Yaskawa INFORM job: DEMO_NAIHAN_0625_2PAINT_1.JBI

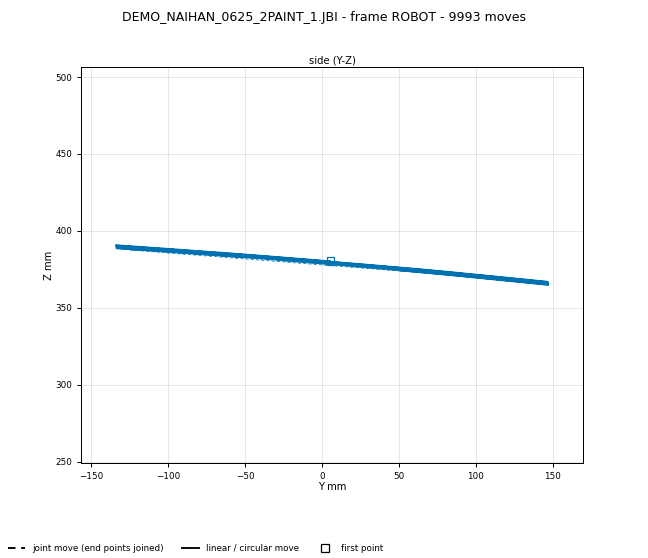
[picture p0: tool path of DEMO_NAIHAN_0625_2PAINT_1.JBI in frame ROBOT, 9993 of 9993 moves have a stored position in this frame; points joined in program order, loops and branches not executed]
/JOB
//NAME DEMO_NAIHAN_0625_2PAINT1
//POS
///NPOS 9993,0,0,0,0,0
///TOOL 1
///USER 0
///POSTYPE ROBOT
///RECTAN
///RCONF 1,0,0,0,1,0,0,0,0,0,0,0,0,0,0,0,0,0,0,0,0,0,0,0
C00000=1015.716,5.571,380.559,-24.182,21.519,-42.786
C00001=1015.718,5.240,380.586,-24.181,21.518,-42.792
C00002=1015.721,4.909,380.612,-24.181,21.519,-42.795
C00003=1015.723,4.578,380.640,-24.180,21.519,-42.799
C00004=1015.725,4.247,380.667,-24.180,21.521,-42.803
C00005=1015.727,3.917,380.694,-24.179,21.520,-42.807
C00006=1015.730,3.604,380.720,-24.179,21.521,-42.810
C00007=1015.732,3.315,380.744,-24.179,21.521,-42.814
C00008=1015.733,3.046,380.766,-24.178,21.522,-42.818
C00009=1015.736,2.783,380.787,-24.177,21.522,-42.823
C00010=1015.737,2.515,380.809,-24.177,21.522,-42.827
C00011=1015.740,2.226,380.832,-24.176,21.523,-42.831
C00012=1015.741,1.915,380.858,-24.176,21.523,-42.834
C00013=1015.744,1.584,380.885,-24.175,21.523,-42.838
C00014=1015.746,1.250,380.912,-24.175,21.524,-42.842
C00015=1015.749,0.917,380.940,-24.174,21.525,-42.846
C00016=1015.750,0.582,380.967,-24.173,21.525,-42.851
C00017=1015.752,0.246,380.994,-24.173,21.525,-42.855
C00018=1015.754,-0.092,381.021,-24.172,21.526,-42.858
C00019=1015.756,-0.430,381.049,-24.172,21.526,-42.864
C00020=1015.759,-0.771,381.077,-24.171,21.526,-42.867
C00021=1015.761,-1.112,381.105,-24.170,21.527,-42.873
C00022=1015.763,-1.455,381.132,-24.170,21.527,-42.877
C00023=1015.766,-1.801,381.161,-24.169,21.528,-42.880
C00024=1015.768,-2.146,381.188,-24.169,21.528,-42.886
C00025=1015.770,-2.495,381.217,-24.168,21.529,-42.890
C00026=1015.772,-2.845,381.245,-24.167,21.529,-42.895
C00027=1015.774,-3.196,381.274,-24.167,21.529,-42.899
C00028=1015.776,-3.549,381.302,-24.166,21.529,-42.904
C00029=1015.778,-3.903,381.331,-24.166,21.531,-42.908
C00030=1015.780,-4.260,381.360,-24.165,21.530,-42.913
C00031=1015.782,-4.622,381.389,-24.164,21.531,-42.919
C00032=1015.784,-4.988,381.419,-24.164,21.532,-42.923
C00033=1015.787,-5.358,381.448,-24.163,21.532,-42.928
C00034=1015.789,-5.732,381.479,-24.163,21.533,-42.932
C00035=1015.791,-6.107,381.510,-24.162,21.533,-42.937
C00036=1015.793,-6.483,381.540,-24.161,21.533,-42.941
C00037=1015.795,-6.858,381.571,-24.160,21.534,-42.947
C00038=1015.797,-7.229,381.601,-24.160,21.534,-42.952
C00039=1015.798,-7.598,381.630,-24.159,21.535,-42.956
C00040=1015.801,-7.964,381.660,-24.158,21.535,-42.961
C00041=1015.802,-8.327,381.689,-24.158,21.536,-42.967
C00042=1015.804,-8.690,381.719,-24.157,21.536,-42.971
C00043=1015.806,-9.053,381.748,-24.156,21.536,-42.976
C00044=1015.808,-9.416,381.776,-24.156,21.537,-42.982
C00045=1015.810,-9.778,381.806,-24.155,21.538,-42.985
C00046=1015.811,-10.139,381.835,-24.154,21.538,-42.991
C00047=1015.814,-10.500,381.865,-24.154,21.539,-42.995
C00048=1015.815,-10.860,381.893,-24.153,21.539,-43.000
C00049=1015.816,-11.219,381.922,-24.152,21.539,-43.006
C00050=1015.819,-11.577,381.950,-24.152,21.540,-43.009
C00051=1015.821,-11.933,381.980,-24.151,21.540,-43.014
C00052=1015.822,-12.288,382.008,-24.151,21.541,-43.019
C00053=1015.823,-12.641,382.036,-24.150,21.541,-43.024
C00054=1015.825,-12.993,382.065,-24.149,21.542,-43.028
C00055=1015.826,-13.344,382.093,-24.149,21.542,-43.033
C00056=1015.828,-13.692,382.121,-24.148,21.543,-43.037
C00057=1015.830,-14.038,382.149,-24.147,21.543,-43.042
C00058=1015.831,-14.383,382.176,-24.147,21.544,-43.046
C00059=1015.832,-14.725,382.203,-24.146,21.544,-43.052
C00060=1015.834,-15.065,382.230,-24.146,21.544,-43.055
C00061=1015.836,-15.402,382.257,-24.145,21.545,-43.061
C00062=1015.837,-15.739,382.285,-24.145,21.546,-43.065
C00063=1015.838,-16.075,382.311,-24.144,21.546,-43.070
C00064=1015.840,-16.408,382.337,-24.143,21.546,-43.074
C00065=1015.841,-16.742,382.364,-24.142,21.547,-43.079
C00066=1015.842,-17.075,382.391,-24.142,21.547,-43.083
C00067=1015.843,-17.409,382.417,-24.141,21.547,-43.088
C00068=1015.845,-17.742,382.444,-24.141,21.548,-43.092
C00069=1015.846,-18.107,382.474,-24.140,21.549,-43.100
C00070=1015.847,-18.329,382.491,-24.139,21.548,-43.103
C00071=1015.848,-18.576,382.510,-24.139,21.549,-43.105
C00072=1015.849,-18.837,382.531,-24.139,21.550,-43.107
C00073=1015.850,-19.099,382.552,-24.139,21.550,-43.109
C00074=1015.851,-19.347,382.573,-24.138,21.550,-43.112
C00075=1015.852,-19.764,382.605,-24.137,21.550,-43.118
C00076=1015.853,-19.936,382.619,-24.137,21.551,-43.122
C00077=1015.854,-20.269,382.646,-24.136,21.551,-43.127
C00078=1015.855,-20.602,382.672,-24.136,21.552,-43.131
C00079=1015.856,-20.934,382.698,-24.135,21.553,-43.135
C00080=1015.857,-21.267,382.725,-24.134,21.552,-43.140
C00081=1015.859,-21.599,382.751,-24.134,21.553,-43.144
C00082=1015.860,-21.933,382.777,-24.133,21.554,-43.149
C00083=1015.861,-22.265,382.804,-24.133,21.554,-43.153
C00084=1015.862,-22.598,382.831,-24.132,21.554,-43.158
C00085=1015.862,-22.930,382.857,-24.131,21.556,-43.162
C00086=1015.864,-23.264,382.883,-24.131,21.555,-43.168
C00087=1015.864,-23.596,382.909,-24.130,21.556,-43.171
C00088=1015.866,-23.929,382.936,-24.129,21.556,-43.177
C00089=1015.866,-24.262,382.962,-24.129,21.557,-43.181
C00090=1015.868,-24.595,382.989,-24.128,21.557,-43.186
C00091=1015.868,-24.928,383.015,-24.128,21.558,-43.190
C00092=1015.869,-25.260,383.041,-24.127,21.558,-43.195
C00093=1015.870,-25.594,383.067,-24.126,21.559,-43.199
C00094=1015.871,-25.926,383.094,-24.126,21.559,-43.204
C00095=1015.871,-26.259,383.120,-24.125,21.559,-43.208
C00096=1015.873,-26.592,383.147,-24.124,21.560,-43.214
C00097=1015.874,-26.924,383.172,-24.124,21.560,-43.217
C00098=1015.875,-27.256,383.198,-24.123,21.560,-43.223
C00099=1015.875,-27.589,383.225,-24.123,21.562,-43.227
C00100=1015.877,-27.922,383.251,-24.122,21.562,-43.232
C00101=1015.877,-28.255,383.277,-24.121,21.562,-43.236
C00102=1015.878,-28.587,383.303,-24.120,21.562,-43.241
C00103=1015.878,-28.920,383.330,-24.120,21.563,-43.245
C00104=1015.879,-29.253,383.355,-24.119,21.563,-43.250
C00105=1015.879,-29.586,383.381,-24.119,21.564,-43.254
C00106=1015.881,-29.918,383.408,-24.118,21.565,-43.260
C00107=1015.882,-30.252,383.434,-24.118,21.565,-43.264
C00108=1015.882,-30.584,383.460,-24.117,21.565,-43.269
C00109=1015.883,-30.917,383.486,-24.116,21.566,-43.273
C00110=1015.883,-31.250,383.512,-24.116,21.566,-43.278
C00111=1015.884,-31.582,383.538,-24.115,21.567,-43.282
C00112=1015.884,-31.915,383.565,-24.114,21.567,-43.287
C00113=1015.885,-32.248,383.590,-24.114,21.568,-43.291
C00114=1015.885,-32.581,383.617,-24.113,21.568,-43.296
C00115=1015.886,-32.914,383.643,-24.113,21.569,-43.301
C00116=1015.886,-33.247,383.668,-24.112,21.569,-43.306
C00117=1015.886,-33.579,383.694,-24.111,21.570,-43.310
C00118=1015.887,-33.912,383.721,-24.111,21.570,-43.315
C00119=1015.888,-34.245,383.746,-24.110,21.571,-43.319
C00120=1015.888,-34.577,383.772,-24.109,21.571,-43.324
C00121=1015.889,-34.910,383.799,-24.109,21.572,-43.328
C00122=1015.889,-35.243,383.824,-24.108,21.572,-43.334
C00123=1015.889,-35.575,383.850,-24.108,21.573,-43.337
C00124=1015.890,-35.908,383.876,-24.107,21.573,-43.343
C00125=1015.890,-36.241,383.902,-24.107,21.574,-43.347
C00126=1015.890,-36.573,383.928,-24.106,21.574,-43.352
C00127=1015.891,-36.905,383.954,-24.105,21.574,-43.357
C00128=1015.892,-37.239,383.979,-24.105,21.575,-43.361
C00129=1015.891,-37.571,384.005,-24.104,21.575,-43.366
C00130=1015.892,-37.903,384.031,-24.103,21.576,-43.371
C00131=1015.893,-38.236,384.057,-24.102,21.576,-43.376
C00132=1015.892,-38.569,384.083,-24.102,21.577,-43.380
C00133=1015.892,-38.902,384.109,-24.101,21.577,-43.385
C00134=1015.892,-39.235,384.134,-24.101,21.578,-43.389
C00135=1015.893,-39.567,384.161,-24.100,21.578,-43.394
C00136=1015.893,-39.899,384.186,-24.100,21.579,-43.398
C00137=1015.894,-40.233,384.212,-24.099,21.579,-43.404
C00138=1015.893,-40.565,384.237,-24.098,21.580,-43.409
C00139=1015.894,-40.897,384.264,-24.098,21.580,-43.413
C00140=1015.894,-41.230,384.289,-24.097,21.580,-43.418
C00141=1015.894,-41.562,384.314,-24.096,21.582,-43.422
C00142=1015.894,-41.895,384.341,-24.096,21.582,-43.427
C00143=1015.894,-42.228,384.366,-24.095,21.582,-43.431
C00144=1015.893,-42.561,384.392,-24.094,21.583,-43.437
C00145=1015.894,-42.893,384.418,-24.094,21.583,-43.442
C00146=1015.894,-43.226,384.443,-24.093,21.583,-43.446
C00147=1015.894,-43.558,384.469,-24.092,21.584,-43.451
C00148=1015.894,-43.890,384.494,-24.092,21.585,-43.455
C00149=1015.894,-44.223,384.520,-24.091,21.585,-43.461
C00150=1015.894,-44.556,384.546,-24.091,21.586,-43.465
C00151=1015.894,-44.888,384.571,-24.090,21.586,-43.470
C00152=1015.894,-45.221,384.596,-24.089,21.586,-43.475
C00153=1015.893,-45.554,384.622,-24.089,21.587,-43.479
C00154=1015.893,-45.886,384.647,-24.088,21.588,-43.485
C00155=1015.893,-46.219,384.673,-24.088,21.588,-43.488
C00156=1015.893,-46.551,384.699,-24.087,21.588,-43.494
C00157=1015.894,-46.884,384.724,-24.086,21.590,-43.498
C00158=1015.893,-47.216,384.750,-24.086,21.589,-43.503
C00159=1015.893,-47.548,384.776,-24.085,21.589,-43.508
C00160=1015.892,-47.881,384.800,-24.084,21.591,-43.512
C00161=1015.892,-48.213,384.826,-24.083,21.591,-43.518
C00162=1015.891,-48.546,384.852,-24.083,21.592,-43.522
C00163=1015.892,-48.879,384.877,-24.082,21.592,-43.527
C00164=1015.891,-49.211,384.902,-24.081,21.592,-43.532
C00165=1015.891,-49.543,384.928,-24.081,21.593,-43.536
C00166=1015.891,-49.876,384.953,-24.080,21.593,-43.542
C00167=1015.891,-50.208,384.979,-24.080,21.595,-43.546
C00168=1015.890,-50.540,385.004,-24.079,21.594,-43.551
C00169=1015.890,-50.873,385.029,-24.079,21.595,-43.555
C00170=1015.890,-51.205,385.055,-24.078,21.596,-43.560
C00171=1015.890,-51.537,385.080,-24.077,21.596,-43.566
C00172=1015.889,-51.870,385.105,-24.077,21.597,-43.570
C00173=1015.888,-52.203,385.131,-24.076,21.597,-43.575
C00174=1015.888,-52.535,385.156,-24.075,21.597,-43.579
C00175=1015.887,-52.867,385.181,-24.075,21.598,-43.584
C00176=1015.887,-53.200,385.206,-24.074,21.598,-43.589
C00177=1015.886,-53.532,385.231,-24.074,21.600,-43.594
C00178=1015.886,-53.864,385.257,-24.073,21.599,-43.599
C00179=1015.885,-54.196,385.282,-24.072,21.600,-43.603
C00180=1015.885,-54.528,385.307,-24.072,21.601,-43.608
C00181=1015.884,-54.860,385.332,-24.071,21.601,-43.613
C00182=1015.884,-55.193,385.357,-24.070,21.602,-43.618
C00183=1015.882,-55.526,385.383,-24.070,21.602,-43.623
C00184=1015.882,-55.859,385.408,-24.069,21.603,-43.627
C00185=1015.882,-56.191,385.434,-24.068,21.603,-43.632
C00186=1015.881,-56.524,385.458,-24.068,21.603,-43.637
C00187=1015.880,-56.858,385.484,-24.067,21.605,-43.642
C00188=1015.880,-57.191,385.509,-24.066,21.604,-43.647
C00189=1015.879,-57.524,385.534,-24.066,21.605,-43.652
C00190=1015.878,-57.858,385.559,-24.065,21.606,-43.656
C00191=1015.877,-58.193,385.584,-24.064,21.606,-43.662
C00192=1015.876,-58.527,385.610,-24.064,21.607,-43.666
C00193=1015.876,-58.862,385.635,-24.063,21.607,-43.671
C00194=1015.875,-59.197,385.660,-24.062,21.608,-43.676
C00195=1015.874,-59.533,385.686,-24.062,21.608,-43.680
C00196=1015.874,-59.869,385.711,-24.061,21.609,-43.686
C00197=1015.873,-60.206,385.736,-24.060,21.609,-43.691
C00198=1015.872,-60.543,385.761,-24.060,21.610,-43.695
C00199=1015.871,-60.880,385.787,-24.059,21.610,-43.700
C00200=1015.870,-61.217,385.812,-24.059,21.611,-43.706
C00201=1015.869,-61.555,385.837,-24.058,21.611,-43.710
C00202=1015.868,-61.894,385.863,-24.057,21.612,-43.715
C00203=1015.867,-62.232,385.888,-24.057,21.612,-43.720
C00204=1015.867,-62.571,385.914,-24.056,21.614,-43.725
C00205=1015.865,-62.911,385.939,-24.055,21.613,-43.730
C00206=1015.864,-63.251,385.965,-24.055,21.614,-43.735
C00207=1015.863,-63.592,385.990,-24.054,21.615,-43.739
C00208=1015.862,-63.933,386.016,-24.053,21.616,-43.745
C00209=1015.861,-64.273,386.041,-24.053,21.615,-43.750
C00210=1015.860,-64.614,386.067,-24.052,21.617,-43.754
C00211=1015.859,-64.956,386.092,-24.051,21.617,-43.759
C00212=1015.857,-65.298,386.118,-24.051,21.618,-43.765
C00213=1015.857,-65.640,386.144,-24.050,21.617,-43.770
C00214=1015.855,-65.983,386.169,-24.050,21.619,-43.774
C00215=1015.854,-66.325,386.195,-24.049,21.619,-43.780
C00216=1015.853,-66.667,386.220,-24.048,21.620,-43.785
C00217=1015.852,-67.011,386.246,-24.048,21.620,-43.789
C00218=1015.850,-67.354,386.271,-24.047,21.621,-43.795
C00219=1015.849,-67.697,386.297,-24.046,21.621,-43.800
C00220=1015.848,-68.041,386.323,-24.045,21.622,-43.805
C00221=1015.846,-68.384,386.348,-24.045,21.622,-43.809
C00222=1015.845,-68.728,386.373,-24.044,21.623,-43.815
C00223=1015.844,-69.072,386.399,-24.043,21.623,-43.820
C00224=1015.843,-69.416,386.425,-24.043,21.624,-43.824
C00225=1015.841,-69.759,386.450,-24.042,21.624,-43.829
C00226=1015.840,-70.104,386.475,-24.041,21.625,-43.835
C00227=1015.838,-70.448,386.501,-24.041,21.625,-43.840
C00228=1015.837,-70.792,386.527,-24.040,21.626,-43.844
C00229=1015.835,-71.136,386.552,-24.040,21.627,-43.850
C00230=1015.834,-71.481,386.577,-24.039,21.627,-43.855
C00231=1015.832,-71.825,386.603,-24.038,21.628,-43.861
C00232=1015.830,-72.168,386.628,-24.038,21.628,-43.865
C00233=1015.829,-72.512,386.654,-24.037,21.629,-43.870
C00234=1015.827,-72.856,386.679,-24.036,21.629,-43.875
C00235=1015.826,-73.200,386.705,-24.035,21.630,-43.881
C00236=1015.824,-73.544,386.729,-24.035,21.630,-43.885
C00237=1015.823,-73.888,386.755,-24.034,21.631,-43.890
C00238=1015.821,-74.232,386.780,-24.033,21.632,-43.896
C00239=1015.820,-74.575,386.806,-24.033,21.632,-43.901
C00240=1015.818,-74.919,386.831,-24.032,21.633,-43.905
C00241=1015.816,-75.262,386.857,-24.031,21.633,-43.911
C00242=1015.814,-75.605,386.882,-24.031,21.634,-43.916
C00243=1015.812,-75.949,386.907,-24.030,21.634,-43.920
C00244=1015.810,-76.291,386.932,-24.030,21.635,-43.926
C00245=1015.809,-76.634,386.957,-24.029,21.635,-43.931
C00246=1015.807,-76.976,386.983,-24.028,21.636,-43.936
C00247=1015.805,-77.318,387.008,-24.028,21.636,-43.940
C00248=1015.804,-77.661,387.032,-24.027,21.637,-43.946
C00249=1015.801,-78.002,387.058,-24.026,21.637,-43.951
C00250=1015.800,-78.344,387.083,-24.026,21.639,-43.955
C00251=1015.798,-78.685,387.108,-24.025,21.638,-43.960
C00252=1015.796,-79.026,387.133,-24.024,21.639,-43.966
C00253=1015.794,-79.366,387.157,-24.023,21.639,-43.971
C00254=1015.792,-79.707,387.183,-24.023,21.641,-43.975
C00255=1015.790,-80.046,387.208,-24.022,21.641,-43.981
C00256=1015.788,-80.386,387.233,-24.021,21.641,-43.986
C00257=1015.786,-80.724,387.257,-24.021,21.643,-43.990
C00258=1015.784,-81.064,387.281,-24.020,21.643,-43.995
C00259=1015.782,-81.402,387.306,-24.020,21.643,-44.001
C00260=1015.780,-81.739,387.331,-24.019,21.644,-44.005
C00261=1015.778,-82.077,387.356,-24.018,21.645,-44.010
C00262=1015.776,-82.414,387.380,-24.018,21.645,-44.016
C00263=1015.773,-82.750,387.405,-24.017,21.645,-44.021
C00264=1015.771,-83.086,387.429,-24.016,21.646,-44.025
C00265=1015.769,-83.422,387.453,-24.016,21.647,-44.031
C00266=1015.767,-83.758,387.477,-24.015,21.647,-44.036
C00267=1015.765,-84.093,387.502,-24.015,21.648,-44.040
C00268=1015.763,-84.426,387.527,-24.014,21.648,-44.045
C00269=1015.760,-84.777,387.552,-24.013,21.649,-44.051
C00270=1015.758,-85.174,387.581,-24.012,21.650,-44.056
C00271=1015.757,-85.386,387.597,-24.012,21.649,-44.060
C00272=1015.755,-85.600,387.612,-24.012,21.649,-44.062
C00273=1015.752,-86.008,387.642,-24.011,21.650,-44.067
C00274=1015.750,-86.367,387.668,-24.010,21.651,-44.073
C00275=1015.747,-86.697,387.692,-24.009,21.652,-44.078
C00276=1015.745,-87.019,387.715,-24.009,21.652,-44.082
C00277=1015.743,-87.336,387.738,-24.008,21.653,-44.088
C00278=1015.741,-87.648,387.760,-24.007,21.653,-44.093
C00279=1015.738,-87.959,387.783,-24.007,21.654,-44.097
C00280=1015.736,-88.271,387.806,-24.006,21.654,-44.102
C00281=1015.734,-88.590,387.828,-24.006,21.655,-44.106
C00282=1015.731,-88.961,387.855,-24.005,21.656,-44.114
C00283=1015.729,-89.181,387.871,-24.004,21.656,-44.117
C00284=1015.728,-89.414,387.888,-24.004,21.656,-44.119
C00285=1015.726,-89.652,387.905,-24.004,21.656,-44.121
C00286=1015.725,-89.884,387.922,-24.004,21.657,-44.123
C00287=1015.721,-90.290,387.951,-24.003,21.658,-44.130
C00288=1015.718,-90.628,387.975,-24.002,21.658,-44.136
C00289=1015.717,-90.957,387.999,-24.001,21.659,-44.141
C00290=1015.714,-91.287,388.023,-24.001,21.660,-44.145
C00291=1015.711,-91.615,388.047,-24.000,21.660,-44.150
C00292=1015.709,-91.943,388.071,-23.999,21.660,-44.156
C00293=1015.706,-92.272,388.093,-23.999,21.661,-44.160
C00294=1015.703,-92.599,388.118,-23.998,21.662,-44.165
C00295=1015.701,-92.925,388.140,-23.998,21.662,-44.169
C00296=1015.698,-93.252,388.164,-23.997,21.663,-44.175
C00297=1015.696,-93.578,388.188,-23.996,21.663,-44.180
C00298=1015.693,-93.902,388.211,-23.996,21.664,-44.184
C00299=1015.690,-94.226,388.234,-23.995,21.664,-44.189
C00300=1015.688,-94.551,388.258,-23.994,21.665,-44.193
C00301=1015.685,-94.875,388.281,-23.994,21.666,-44.199
C00302=1015.681,-95.198,388.304,-23.993,21.666,-44.204
C00303=1015.679,-95.521,388.327,-23.993,21.666,-44.207
C00304=1015.676,-95.842,388.350,-23.992,21.667,-44.213
C00305=1015.674,-96.165,388.373,-23.991,21.668,-44.217
C00306=1015.670,-96.487,388.396,-23.991,21.668,-44.222
C00307=1015.668,-96.808,388.419,-23.990,21.669,-44.226
C00308=1015.665,-97.129,388.442,-23.989,21.669,-44.231
C00309=1015.662,-97.450,388.465,-23.989,21.670,-44.236
C00310=1015.660,-97.771,388.488,-23.988,21.670,-44.241
C00311=1015.656,-98.092,388.511,-23.987,21.670,-44.246
C00312=1015.654,-98.412,388.534,-23.987,21.672,-44.250
C00313=1015.650,-98.733,388.557,-23.986,21.671,-44.255
C00314=1015.648,-99.055,388.579,-23.986,21.673,-44.260
C00315=1015.645,-99.376,388.602,-23.985,21.673,-44.265
C00316=1015.641,-99.697,388.625,-23.985,21.673,-44.268
C00317=1015.639,-100.019,388.647,-23.984,21.674,-44.274
C00318=1015.635,-100.341,388.671,-23.983,21.675,-44.278
C00319=1015.632,-100.663,388.694,-23.983,21.675,-44.283
C00320=1015.630,-100.985,388.717,-23.982,21.676,-44.287
C00321=1015.626,-101.309,388.740,-23.981,21.676,-44.292
C00322=1015.623,-101.632,388.763,-23.981,21.677,-44.298
C00323=1015.620,-101.956,388.786,-23.980,21.677,-44.302
C00324=1015.617,-102.282,388.808,-23.980,21.678,-44.307
C00325=1015.614,-102.606,388.832,-23.979,21.679,-44.311
C00326=1015.610,-102.932,388.855,-23.978,21.679,-44.316
C00327=1015.607,-103.258,388.878,-23.978,21.680,-44.320
C00328=1015.604,-103.584,388.901,-23.977,21.680,-44.326
C00329=1015.601,-103.912,388.924,-23.976,21.681,-44.331
C00330=1015.597,-104.239,388.947,-23.976,21.681,-44.335
C00331=1015.594,-104.567,388.970,-23.975,21.681,-44.340
C00332=1015.591,-104.894,388.994,-23.975,21.683,-44.344
C00333=1015.587,-105.223,389.017,-23.974,21.683,-44.350
C00334=1015.584,-105.552,389.040,-23.974,21.684,-44.354
C00335=1015.580,-105.880,389.064,-23.973,21.684,-44.359
C00336=1015.577,-106.209,389.087,-23.972,21.685,-44.365
C00337=1015.573,-106.538,389.110,-23.972,21.685,-44.368
C00338=1015.570,-106.867,389.133,-23.971,21.685,-44.374
C00339=1015.566,-107.196,389.156,-23.971,21.687,-44.378
C00340=1015.562,-107.525,389.180,-23.970,21.687,-44.383
C00341=1015.558,-107.855,389.203,-23.969,21.687,-44.388
C00342=1015.555,-108.184,389.226,-23.969,21.688,-44.392
C00343=1015.551,-108.512,389.249,-23.968,21.689,-44.398
C00344=1015.548,-108.841,389.272,-23.967,21.689,-44.402
C00345=1015.544,-109.170,389.295,-23.967,21.689,-44.407
C00346=1015.540,-109.499,389.319,-23.966,21.690,-44.412
C00347=1015.537,-109.828,389.342,-23.965,21.691,-44.416
C00348=1015.533,-110.158,389.365,-23.965,21.691,-44.422
C00349=1015.530,-110.486,389.388,-23.964,21.692,-44.426
C00350=1015.526,-110.815,389.412,-23.963,21.692,-44.431
C00351=1015.522,-111.144,389.434,-23.963,21.693,-44.436
C00352=1015.518,-111.473,389.458,-23.962,21.693,-44.440
C00353=1015.514,-111.802,389.481,-23.962,21.694,-44.446
C00354=1015.510,-112.130,389.503,-23.961,21.695,-44.449
C00355=1015.506,-112.459,389.527,-23.960,21.695,-44.455
C00356=1015.503,-112.788,389.550,-23.960,21.696,-44.459
C00357=1015.498,-113.116,389.573,-23.959,21.696,-44.464
C00358=1015.494,-113.446,389.596,-23.958,21.697,-44.470
C00359=1015.491,-113.774,389.618,-23.958,21.697,-44.473
C00360=1015.487,-114.102,389.642,-23.957,21.698,-44.479
C00361=1015.482,-114.431,389.664,-23.957,21.699,-44.483
C00362=1015.478,-114.760,389.688,-23.956,21.699,-44.488
C00363=1015.475,-115.088,389.710,-23.956,21.700,-44.492
C00364=1015.471,-115.417,389.734,-23.955,21.700,-44.497
C00365=1015.466,-115.746,389.757,-23.954,21.701,-44.503
C00366=1015.462,-116.074,389.780,-23.954,21.701,-44.507
C00367=1015.458,-116.404,389.803,-23.953,21.701,-44.512
C00368=1015.454,-116.731,389.826,-23.953,21.703,-44.516
C00369=1015.449,-117.060,389.849,-23.952,21.703,-44.521
C00370=1015.447,-117.277,389.864,-23.952,21.704,-44.523
C00371=1015.443,-117.497,389.879,-23.951,21.703,-44.527
C00372=1015.441,-117.717,389.895,-23.951,21.704,-44.531
C00373=1015.437,-118.045,389.917,-23.950,21.705,-44.535
C00374=1015.432,-118.374,389.940,-23.949,21.705,-44.540
C00375=1015.428,-118.702,389.963,-23.949,21.705,-44.545
C00376=1015.423,-119.031,389.986,-23.948,21.707,-44.549
C00377=1015.419,-119.359,390.009,-23.948,21.707,-44.554
C00378=1015.415,-119.688,390.031,-23.947,21.707,-44.558
C00379=1015.410,-120.016,390.054,-23.946,21.708,-44.564
C00380=1015.405,-120.344,390.078,-23.946,21.709,-44.568
C00381=1015.401,-120.673,390.100,-23.945,21.709,-44.573
C00382=1015.397,-121.001,390.123,-23.945,21.710,-44.577
C00383=1015.392,-121.329,390.146,-23.944,21.710,-44.582
C00384=1015.388,-121.658,390.169,-23.944,21.711,-44.586
C00385=1015.383,-121.987,390.192,-23.943,21.711,-44.591
C00386=1015.379,-122.315,390.215,-23.942,21.712,-44.597
C00387=1015.374,-122.642,390.237,-23.942,21.713,-44.601
C00388=1015.369,-122.971,390.260,-23.941,21.713,-44.606
C00389=1015.365,-123.300,390.283,-23.940,21.714,-44.610
C00390=1015.360,-123.628,390.306,-23.940,21.714,-44.615
C00391=1015.355,-123.957,390.328,-23.939,21.715,-44.620
C00392=1015.351,-124.284,390.351,-23.939,21.715,-44.625
C00393=1015.346,-124.612,390.374,-23.938,21.716,-44.628
C00394=1015.341,-124.941,390.396,-23.937,21.717,-44.634
C00395=1015.336,-125.269,390.420,-23.937,21.717,-44.638
C00396=1015.331,-125.597,390.441,-23.936,21.717,-44.643
C00397=1015.326,-125.926,390.465,-23.936,21.719,-44.647
C00398=1015.321,-126.254,390.487,-23.935,21.719,-44.652
C00399=1015.317,-126.581,390.510,-23.935,21.720,-44.657
C00400=1015.311,-126.909,390.533,-23.934,21.720,-44.662
C00401=1015.307,-127.238,390.555,-23.933,21.720,-44.667
C00402=1015.302,-127.566,390.578,-23.933,21.721,-44.671
C00403=1015.297,-127.895,390.601,-23.932,21.721,-44.676
C00404=1015.291,-128.223,390.624,-23.931,21.722,-44.680
C00405=1015.286,-128.551,390.646,-23.931,21.723,-44.686
C00406=1015.281,-128.879,390.669,-23.930,21.723,-44.689
C00407=1015.276,-129.207,390.692,-23.929,21.723,-44.695
C00408=1015.271,-129.535,390.714,-23.929,21.725,-44.699
C00409=1015.267,-129.864,390.737,-23.928,21.724,-44.704
C00410=1015.261,-130.192,390.759,-23.928,21.726,-44.708
C00411=1015.256,-130.520,390.782,-23.927,21.726,-44.713
C00412=1015.250,-130.848,390.804,-23.927,21.726,-44.717
C00413=1015.245,-131.176,390.827,-23.926,21.727,-44.723
C00414=1015.240,-131.504,390.849,-23.926,21.728,-44.726
C00415=1015.235,-131.832,390.873,-23.925,21.728,-44.732
C00416=1015.230,-132.160,390.895,-23.924,21.729,-44.736
C00417=1015.224,-132.488,390.918,-23.924,21.729,-44.741
C00418=1015.219,-132.816,390.940,-23.923,21.730,-44.745
C00419=1015.213,-133.144,390.963,-23.922,21.731,-44.750
C00420=1015.208,-133.472,390.986,-23.922,21.731,-44.754
C00421=1015.202,-133.800,391.008,-23.921,21.731,-44.759
C00422=1015.197,-134.128,391.031,-23.921,21.732,-44.763
C00423=1015.615,-134.098,390.769,-23.921,21.732,-44.763
C00424=1015.621,-133.770,390.746,-23.921,21.731,-44.759
C00425=1015.626,-133.441,390.725,-23.922,21.731,-44.754
C00426=1015.631,-133.114,390.702,-23.922,21.731,-44.750
C00427=1015.636,-132.786,390.680,-23.923,21.730,-44.745
C00428=1015.642,-132.458,390.657,-23.924,21.729,-44.741
C00429=1015.647,-132.130,390.635,-23.924,21.729,-44.736
C00430=1015.651,-131.802,390.613,-23.925,21.728,-44.732
C00431=1015.656,-131.474,390.590,-23.926,21.728,-44.726
C00432=1015.662,-131.146,390.567,-23.926,21.727,-44.723
C00433=1015.667,-130.818,390.545,-23.927,21.726,-44.717
C00434=1015.671,-130.490,390.523,-23.927,21.726,-44.713
C00435=1015.676,-130.161,390.500,-23.928,21.726,-44.708
C00436=1015.682,-129.833,390.477,-23.928,21.724,-44.704
C00437=1015.687,-129.505,390.456,-23.929,21.725,-44.699
C00438=1015.691,-129.177,390.433,-23.929,21.723,-44.695
C00439=1015.696,-128.849,390.410,-23.930,21.723,-44.689
C00440=1015.702,-128.521,390.388,-23.931,21.723,-44.686
C00441=1015.705,-128.193,390.366,-23.931,21.722,-44.680
C00442=1015.711,-127.865,390.343,-23.932,21.721,-44.676
C00443=1015.715,-127.536,390.320,-23.933,21.721,-44.671
C00444=1015.720,-127.208,390.298,-23.933,21.720,-44.667
C00445=1015.725,-126.880,390.275,-23.934,21.720,-44.662
C00446=1015.730,-126.552,390.252,-23.935,21.720,-44.657
C00447=1015.734,-126.224,390.230,-23.935,21.719,-44.652
C00448=1015.739,-125.896,390.207,-23.936,21.719,-44.647
C00449=1015.744,-125.567,390.185,-23.936,21.717,-44.643
C00450=1015.748,-125.239,390.162,-23.937,21.717,-44.638
C00451=1015.752,-124.911,390.139,-23.937,21.717,-44.634
C00452=1015.758,-124.582,390.117,-23.938,21.716,-44.628
C00453=1015.762,-124.255,390.095,-23.939,21.715,-44.625
C00454=1015.766,-123.926,390.071,-23.939,21.715,-44.620
C00455=1015.771,-123.598,390.050,-23.940,21.714,-44.615
C00456=1015.776,-123.270,390.027,-23.940,21.714,-44.610
C00457=1015.780,-122.941,390.004,-23.941,21.713,-44.606
C00458=1015.784,-122.613,389.981,-23.942,21.713,-44.601
C00459=1015.789,-122.285,389.958,-23.942,21.712,-44.597
C00460=1015.793,-121.956,389.936,-23.943,21.711,-44.591
C00461=1015.797,-121.628,389.913,-23.944,21.711,-44.586
C00462=1015.801,-121.300,389.891,-23.944,21.710,-44.582
C00463=1015.806,-120.972,389.868,-23.945,21.710,-44.577
C00464=1015.810,-120.643,389.845,-23.945,21.709,-44.573
C00465=1015.815,-120.315,389.822,-23.946,21.709,-44.568
C00466=1015.818,-119.986,389.800,-23.946,21.708,-44.564
C00467=1015.823,-119.658,389.777,-23.947,21.707,-44.558
C00468=1015.827,-119.330,389.755,-23.948,21.707,-44.554
C00469=1015.832,-119.001,389.731,-23.948,21.707,-44.549
C00470=1015.836,-118.672,389.709,-23.949,21.705,-44.545
C00471=1015.840,-118.345,389.686,-23.949,21.705,-44.540
C00472=1015.844,-118.016,389.663,-23.950,21.705,-44.535
C00473=1015.848,-117.688,389.640,-23.951,21.704,-44.531
C00474=1015.852,-117.359,389.618,-23.951,21.704,-44.525
C00475=1015.856,-117.030,389.595,-23.952,21.703,-44.521
C00476=1015.860,-116.702,389.572,-23.953,21.703,-44.516
C00477=1015.864,-116.373,389.550,-23.953,21.701,-44.512
C00478=1015.868,-116.045,389.527,-23.954,21.701,-44.507
C00479=1015.872,-115.716,389.504,-23.954,21.701,-44.503
C00480=1015.876,-115.387,389.481,-23.955,21.700,-44.497
C00481=1015.880,-115.059,389.458,-23.956,21.700,-44.492
C00482=1015.884,-114.730,389.435,-23.956,21.699,-44.488
C00483=1015.887,-114.402,389.412,-23.957,21.699,-44.483
C00484=1015.892,-114.073,389.389,-23.957,21.698,-44.479
C00485=1015.895,-113.744,389.366,-23.958,21.697,-44.473
C00486=1015.899,-113.416,389.344,-23.958,21.697,-44.470
C00487=1015.903,-113.087,389.320,-23.959,21.696,-44.464
C00488=1015.907,-112.758,389.297,-23.960,21.696,-44.459
C00489=1015.910,-112.430,389.275,-23.960,21.695,-44.455
C00490=1015.914,-112.101,389.252,-23.961,21.695,-44.449
C00491=1015.917,-111.772,389.229,-23.962,21.694,-44.446
C00492=1015.921,-111.443,389.206,-23.962,21.693,-44.440
C00493=1015.926,-111.115,389.183,-23.963,21.693,-44.436
C00494=1015.929,-110.786,389.160,-23.963,21.692,-44.431
C00495=1015.932,-110.457,389.137,-23.964,21.692,-44.426
C00496=1015.936,-110.128,389.114,-23.965,21.691,-44.422
C00497=1015.939,-109.799,389.091,-23.965,21.691,-44.416
C00498=1015.943,-109.470,389.067,-23.966,21.690,-44.412
C00499=1015.947,-109.141,389.044,-23.967,21.689,-44.407
C00500=1015.950,-108.812,389.021,-23.967,21.689,-44.402
C00501=1015.953,-108.483,388.998,-23.968,21.689,-44.398
C00502=1015.957,-108.154,388.975,-23.969,21.688,-44.392
C00503=1015.961,-107.825,388.952,-23.969,21.687,-44.388
C00504=1015.964,-107.496,388.930,-23.970,21.687,-44.383
C00505=1015.968,-107.168,388.906,-23.971,21.687,-44.378
C00506=1015.971,-106.838,388.883,-23.971,21.685,-44.374
C00507=1015.974,-106.510,388.860,-23.972,21.685,-44.368
C00508=1015.978,-106.180,388.837,-23.972,21.685,-44.365
C00509=1015.981,-105.851,388.813,-23.973,21.684,-44.359
C00510=1015.984,-105.523,388.790,-23.974,21.684,-44.354
C00511=1015.987,-105.194,388.767,-23.974,21.683,-44.350
C00512=1015.991,-104.865,388.744,-23.975,21.683,-44.344
C00513=1015.994,-104.537,388.721,-23.975,21.681,-44.340
C00514=1015.997,-104.210,388.698,-23.976,21.681,-44.335
C00515=1016.001,-103.882,388.675,-23.976,21.681,-44.331
C00516=1016.004,-103.555,388.652,-23.977,21.680,-44.326
C00517=1016.007,-103.229,388.629,-23.978,21.680,-44.320
C00518=1016.010,-102.903,388.605,-23.978,21.679,-44.316
C00519=1016.013,-102.577,388.583,-23.979,21.679,-44.311
C00520=1016.016,-102.252,388.560,-23.980,21.678,-44.307
C00521=1016.019,-101.927,388.537,-23.980,21.677,-44.302
C00522=1016.022,-101.603,388.513,-23.981,21.677,-44.298
C00523=1016.025,-101.280,388.491,-23.981,21.676,-44.292
C00524=1016.028,-100.957,388.468,-23.982,21.676,-44.287
C00525=1016.031,-100.635,388.445,-23.983,21.675,-44.283
C00526=1016.034,-100.312,388.422,-23.983,21.675,-44.278
C00527=1016.037,-99.990,388.399,-23.984,21.674,-44.274
C00528=1016.040,-99.668,388.377,-23.985,21.673,-44.268
C00529=1016.043,-99.347,388.354,-23.985,21.673,-44.265
C00530=1016.045,-99.026,388.331,-23.986,21.673,-44.260
C00531=1016.048,-98.705,388.308,-23.986,21.671,-44.255
C00532=1016.051,-98.384,388.286,-23.987,21.672,-44.250
C00533=1016.054,-98.063,388.263,-23.987,21.670,-44.246
C00534=1016.057,-97.743,388.240,-23.988,21.670,-44.241
C00535=1016.060,-97.421,388.217,-23.989,21.670,-44.236
C00536=1016.062,-97.100,388.194,-23.989,21.669,-44.231
C00537=1016.065,-96.779,388.171,-23.990,21.669,-44.226
C00538=1016.068,-96.458,388.148,-23.991,21.668,-44.222
C00539=1016.071,-96.136,388.125,-23.991,21.668,-44.217
C00540=1016.073,-95.814,388.102,-23.992,21.667,-44.213
C00541=1016.076,-95.492,388.080,-23.993,21.666,-44.207
C00542=1016.078,-95.169,388.056,-23.993,21.666,-44.204
C00543=1016.081,-94.846,388.033,-23.994,21.666,-44.199
C00544=1016.083,-94.522,388.010,-23.994,21.665,-44.193
C00545=1016.086,-94.198,387.987,-23.995,21.664,-44.189
C00546=1016.089,-93.874,387.964,-23.996,21.664,-44.184
C00547=1016.091,-93.549,387.941,-23.996,21.663,-44.180
C00548=1016.094,-93.223,387.918,-23.997,21.663,-44.175
C00549=1016.097,-92.897,387.894,-23.998,21.662,-44.169
C00550=1016.099,-92.570,387.871,-23.998,21.662,-44.165
C00551=1016.102,-92.243,387.847,-23.999,21.661,-44.160
C00552=1016.104,-91.915,387.823,-23.999,21.660,-44.156
C00553=1016.106,-91.586,387.800,-24.000,21.660,-44.150
C00554=1016.109,-91.257,387.776,-24.001,21.660,-44.145
C00555=1016.111,-90.929,387.752,-24.001,21.659,-44.141
C00556=1016.114,-90.599,387.729,-24.002,21.658,-44.136
C00557=1016.116,-90.261,387.704,-24.003,21.658,-44.130
C00558=1016.119,-89.855,387.676,-24.004,21.657,-44.123
C00559=1016.121,-89.624,387.659,-24.004,21.656,-44.121
C00560=1016.123,-89.385,387.642,-24.004,21.656,-44.119
C00561=1016.124,-89.152,387.625,-24.004,21.656,-44.117
C00562=1016.126,-88.932,387.609,-24.005,21.656,-44.114
C00563=1016.128,-88.562,387.583,-24.006,21.655,-44.106
C00564=1016.131,-88.243,387.560,-24.006,21.654,-44.102
C00565=1016.133,-87.930,387.537,-24.007,21.654,-44.097
C00566=1016.135,-87.619,387.514,-24.007,21.653,-44.093
C00567=1016.137,-87.308,387.492,-24.008,21.653,-44.088
C00568=1016.139,-86.991,387.470,-24.009,21.652,-44.082
C00569=1016.142,-86.668,387.446,-24.009,21.652,-44.078
C00570=1016.143,-86.339,387.422,-24.010,21.651,-44.073
C00571=1016.146,-85.980,387.396,-24.011,21.650,-44.067
C00572=1016.148,-85.571,387.366,-24.012,21.649,-44.062
C00573=1016.150,-85.357,387.351,-24.012,21.649,-44.060
C00574=1016.151,-85.145,387.336,-24.012,21.650,-44.056
C00575=1016.154,-84.748,387.307,-24.013,21.649,-44.051
C00576=1016.156,-84.398,387.281,-24.014,21.648,-44.045
C00577=1016.159,-84.064,387.257,-24.015,21.648,-44.040
C00578=1016.160,-83.729,387.233,-24.015,21.647,-44.036
C00579=1016.162,-83.394,387.208,-24.016,21.647,-44.031
C00580=1016.164,-83.058,387.184,-24.016,21.646,-44.025
C00581=1016.167,-82.722,387.160,-24.017,21.645,-44.021
C00582=1016.168,-82.386,387.136,-24.018,21.645,-44.016
C00583=1016.170,-82.049,387.111,-24.018,21.645,-44.010
C00584=1016.173,-81.711,387.087,-24.019,21.644,-44.005
C00585=1016.175,-81.374,387.062,-24.020,21.643,-44.001
C00586=1016.177,-81.036,387.037,-24.020,21.643,-43.995
C00587=1016.179,-80.696,387.013,-24.021,21.643,-43.990
C00588=1016.180,-80.357,386.987,-24.021,21.641,-43.986
C00589=1016.182,-80.018,386.963,-24.022,21.641,-43.981
C00590=1016.184,-79.678,386.938,-24.023,21.641,-43.975
C00591=1016.186,-79.338,386.913,-24.023,21.639,-43.971
C00592=1016.188,-78.997,386.888,-24.024,21.639,-43.966
C00593=1016.190,-78.656,386.863,-24.025,21.638,-43.960
C00594=1016.192,-78.315,386.838,-24.026,21.639,-43.955
C00595=1016.194,-77.974,386.814,-24.026,21.637,-43.951
C00596=1016.195,-77.632,386.788,-24.027,21.637,-43.946
C00597=1016.197,-77.291,386.764,-24.028,21.636,-43.940
C00598=1016.199,-76.948,386.738,-24.028,21.636,-43.936
C00599=1016.200,-76.605,386.713,-24.029,21.635,-43.931
C00600=1016.202,-76.263,386.688,-24.030,21.635,-43.926
C00601=1016.203,-75.920,386.663,-24.030,21.634,-43.920
C00602=1016.205,-75.577,386.638,-24.031,21.634,-43.916
C00603=1016.207,-75.234,386.613,-24.031,21.633,-43.911
C00604=1016.209,-74.891,386.587,-24.032,21.633,-43.905
C00605=1016.211,-74.547,386.562,-24.033,21.632,-43.901
C00606=1016.212,-74.204,386.536,-24.033,21.632,-43.896
C00607=1016.214,-73.860,386.511,-24.034,21.631,-43.890
C00608=1016.214,-73.516,386.486,-24.035,21.630,-43.885
C00609=1016.216,-73.172,386.461,-24.035,21.630,-43.881
C00610=1016.218,-72.828,386.435,-24.036,21.629,-43.875
C00611=1016.220,-72.484,386.410,-24.037,21.629,-43.870
C00612=1016.221,-72.140,386.384,-24.038,21.628,-43.865
C00613=1016.223,-71.796,386.360,-24.038,21.628,-43.861
C00614=1016.224,-71.452,386.334,-24.039,21.627,-43.855
C00615=1016.226,-71.108,386.308,-24.040,21.627,-43.850
C00616=1016.227,-70.764,386.282,-24.040,21.626,-43.844
C00617=1016.229,-70.419,386.258,-24.041,21.625,-43.840
C00618=1016.230,-70.075,386.232,-24.041,21.625,-43.835
C00619=1016.231,-69.732,386.206,-24.042,21.624,-43.829
C00620=1016.232,-69.388,386.181,-24.043,21.624,-43.824
C00621=1016.234,-69.043,386.156,-24.043,21.623,-43.820
C00622=1016.235,-68.699,386.130,-24.044,21.623,-43.815
C00623=1016.236,-68.356,386.105,-24.045,21.622,-43.809
C00624=1016.237,-68.012,386.079,-24.045,21.622,-43.805
C00625=1016.240,-67.669,386.053,-24.046,21.621,-43.800
C00626=1016.240,-67.326,386.028,-24.047,21.621,-43.795
C00627=1016.241,-66.983,386.002,-24.048,21.620,-43.789
C00628=1016.243,-66.639,385.977,-24.048,21.620,-43.785
C00629=1016.244,-66.297,385.951,-24.049,21.619,-43.780
C00630=1016.246,-65.954,385.926,-24.050,21.619,-43.774
C00631=1016.246,-65.612,385.901,-24.050,21.617,-43.770
C00632=1016.247,-65.269,385.875,-24.051,21.618,-43.765
C00633=1016.248,-64.928,385.850,-24.051,21.617,-43.759
C00634=1016.249,-64.587,385.823,-24.052,21.617,-43.754
C00635=1016.250,-64.245,385.798,-24.053,21.615,-43.750
C00636=1016.252,-63.904,385.772,-24.053,21.616,-43.745
C00637=1016.252,-63.563,385.748,-24.054,21.615,-43.739
C00638=1016.253,-63.223,385.722,-24.055,21.614,-43.735
C00639=1016.255,-62.884,385.697,-24.055,21.613,-43.730
C00640=1016.256,-62.543,385.671,-24.056,21.614,-43.725
C00641=1016.256,-62.205,385.645,-24.057,21.612,-43.720
C00642=1016.257,-61.865,385.621,-24.057,21.612,-43.715
C00643=1016.259,-61.527,385.595,-24.058,21.611,-43.710
C00644=1016.259,-61.189,385.570,-24.059,21.611,-43.706
C00645=1016.260,-60.852,385.545,-24.059,21.610,-43.700
C00646=1016.261,-60.514,385.519,-24.060,21.610,-43.695
C00647=1016.262,-60.177,385.494,-24.060,21.609,-43.691
C00648=1016.262,-59.841,385.468,-24.061,21.609,-43.686
C00649=1016.264,-59.505,385.443,-24.062,21.608,-43.680
C00650=1016.264,-59.169,385.417,-24.062,21.608,-43.676
C00651=1016.265,-58.834,385.393,-24.063,21.607,-43.671
C00652=1016.266,-58.499,385.367,-24.064,21.607,-43.666
C00653=1016.267,-58.164,385.342,-24.064,21.606,-43.662
C00654=1016.267,-57.830,385.318,-24.065,21.606,-43.656
C00655=1016.268,-57.496,385.292,-24.066,21.605,-43.652
C00656=1016.269,-57.162,385.266,-24.066,21.604,-43.647
C00657=1016.269,-56.829,385.241,-24.067,21.605,-43.642
C00658=1016.269,-56.496,385.216,-24.068,21.603,-43.637
C00659=1016.270,-56.163,385.191,-24.068,21.603,-43.632
C00660=1016.271,-55.830,385.165,-24.069,21.603,-43.627
C00661=1016.272,-55.497,385.141,-24.070,21.602,-43.623
C00662=1016.272,-55.165,385.115,-24.070,21.602,-43.618
C00663=1016.273,-54.833,385.091,-24.071,21.601,-43.613
C00664=1016.273,-54.501,385.065,-24.072,21.601,-43.608
C00665=1016.274,-54.168,385.040,-24.072,21.600,-43.603
C00666=1016.274,-53.835,385.015,-24.073,21.599,-43.599
C00667=1016.275,-53.503,384.989,-24.074,21.600,-43.594
C00668=1016.276,-53.171,384.964,-24.074,21.598,-43.589
C00669=1016.275,-52.838,384.939,-24.075,21.598,-43.584
C00670=1016.276,-52.506,384.914,-24.075,21.597,-43.579
C00671=1016.277,-52.174,384.888,-24.076,21.597,-43.575
C00672=1016.277,-51.842,384.863,-24.077,21.597,-43.570
C00673=1016.278,-51.509,384.838,-24.077,21.596,-43.566
C00674=1016.278,-51.177,384.812,-24.078,21.596,-43.560
C00675=1016.278,-50.845,384.787,-24.079,21.595,-43.555
C00676=1016.279,-50.513,384.762,-24.079,21.594,-43.551
C00677=1016.279,-50.180,384.737,-24.080,21.595,-43.546
C00678=1016.279,-49.848,384.711,-24.080,21.593,-43.542
C00679=1016.279,-49.515,384.686,-24.081,21.593,-43.536
C00680=1016.279,-49.183,384.660,-24.081,21.592,-43.532
C00681=1016.280,-48.850,384.635,-24.082,21.592,-43.527
C00682=1016.280,-48.517,384.609,-24.083,21.592,-43.522
C00683=1016.280,-48.185,384.584,-24.083,21.591,-43.518
C00684=1016.281,-47.853,384.559,-24.084,21.591,-43.512
C00685=1016.281,-47.520,384.534,-24.085,21.589,-43.508
C00686=1016.281,-47.188,384.508,-24.086,21.589,-43.503
C00687=1016.281,-46.855,384.483,-24.086,21.590,-43.498
C00688=1016.281,-46.523,384.457,-24.087,21.588,-43.494
C00689=1016.281,-46.191,384.431,-24.088,21.588,-43.488
C00690=1016.281,-45.858,384.406,-24.088,21.588,-43.485
C00691=1016.282,-45.525,384.380,-24.089,21.587,-43.479
C00692=1016.282,-45.193,384.354,-24.089,21.586,-43.475
C00693=1016.282,-44.860,384.329,-24.090,21.586,-43.470
C00694=1016.282,-44.528,384.304,-24.091,21.586,-43.465
C00695=1016.282,-44.195,384.279,-24.091,21.585,-43.461
C00696=1016.282,-43.862,384.252,-24.092,21.585,-43.455
C00697=1016.282,-43.530,384.227,-24.092,21.584,-43.451
C00698=1016.282,-43.197,384.202,-24.093,21.583,-43.446
C00699=1016.282,-42.865,384.176,-24.094,21.583,-43.442
C00700=1016.281,-42.533,384.150,-24.094,21.583,-43.437
C00701=1016.282,-42.199,384.124,-24.095,21.582,-43.431
C00702=1016.282,-41.867,384.099,-24.096,21.582,-43.427
C00703=1016.282,-41.534,384.072,-24.096,21.582,-43.422
C00704=1016.282,-41.202,384.047,-24.097,21.580,-43.418
C00705=1016.282,-40.869,384.022,-24.098,21.580,-43.413
C00706=1016.281,-40.537,383.995,-24.098,21.580,-43.409
C00707=1016.281,-40.204,383.970,-24.099,21.579,-43.404
C00708=1016.281,-39.872,383.944,-24.100,21.579,-43.398
C00709=1016.281,-39.539,383.918,-24.100,21.578,-43.394
C00710=1016.280,-39.206,383.893,-24.101,21.578,-43.389
C00711=1016.280,-38.874,383.867,-24.101,21.577,-43.385
C00712=1016.280,-38.541,383.841,-24.102,21.577,-43.380
C00713=1016.280,-38.208,383.816,-24.102,21.576,-43.376
C00714=1016.280,-37.875,383.789,-24.103,21.576,-43.371
C00715=1016.279,-37.543,383.763,-24.104,21.575,-43.366
C00716=1016.279,-37.210,383.738,-24.105,21.575,-43.361
C00717=1016.279,-36.878,383.712,-24.105,21.574,-43.357
C00718=1016.278,-36.545,383.685,-24.106,21.574,-43.352
C00719=1016.278,-36.212,383.661,-24.107,21.574,-43.347
C00720=1016.278,-35.880,383.634,-24.107,21.573,-43.343
C00721=1016.277,-35.547,383.608,-24.108,21.573,-43.337
C00722=1016.276,-35.214,383.582,-24.108,21.572,-43.334
C00723=1016.277,-34.882,383.557,-24.109,21.572,-43.328
C00724=1016.276,-34.549,383.530,-24.109,21.571,-43.324
C00725=1016.275,-34.216,383.505,-24.110,21.571,-43.319
C00726=1016.275,-33.884,383.479,-24.111,21.570,-43.315
C00727=1016.274,-33.551,383.452,-24.111,21.570,-43.310
C00728=1016.274,-33.217,383.426,-24.112,21.569,-43.306
C00729=1016.274,-32.885,383.401,-24.113,21.569,-43.301
C00730=1016.274,-32.553,383.374,-24.113,21.568,-43.296
C00731=1016.273,-32.220,383.349,-24.114,21.568,-43.291
C00732=1016.272,-31.887,383.323,-24.114,21.567,-43.287
C00733=1016.272,-31.554,383.296,-24.115,21.567,-43.282
C00734=1016.271,-31.221,383.271,-24.116,21.566,-43.278
C00735=1016.271,-30.889,383.244,-24.116,21.566,-43.273
C00736=1016.270,-30.556,383.218,-24.117,21.565,-43.269
C00737=1016.270,-30.224,383.192,-24.118,21.565,-43.264
C00738=1016.269,-29.891,383.166,-24.118,21.565,-43.260
C00739=1016.268,-29.558,383.140,-24.119,21.564,-43.254
C00740=1016.267,-29.225,383.113,-24.119,21.563,-43.250
C00741=1016.266,-28.892,383.088,-24.120,21.563,-43.245
C00742=1016.266,-28.560,383.061,-24.120,21.562,-43.241
C00743=1016.265,-28.227,383.035,-24.121,21.562,-43.236
C00744=1016.265,-27.895,383.009,-24.122,21.562,-43.232
C00745=1016.264,-27.561,382.983,-24.123,21.562,-43.227
C00746=1016.263,-27.229,382.956,-24.123,21.560,-43.223
C00747=1016.262,-26.896,382.930,-24.124,21.560,-43.217
C00748=1016.261,-26.563,382.904,-24.124,21.560,-43.214
C00749=1016.260,-26.230,382.877,-24.125,21.559,-43.208
C00750=1016.259,-25.898,382.851,-24.126,21.559,-43.204
C00751=1016.259,-25.565,382.825,-24.126,21.559,-43.199
C00752=1016.257,-25.232,382.799,-24.127,21.558,-43.195
C00753=1016.257,-24.899,382.772,-24.128,21.558,-43.190
C00754=1016.256,-24.567,382.746,-24.128,21.557,-43.186
C00755=1016.255,-24.234,382.719,-24.129,21.557,-43.181
C00756=1016.254,-23.901,382.694,-24.129,21.556,-43.177
C00757=1016.253,-23.568,382.667,-24.130,21.556,-43.171
C00758=1016.253,-23.235,382.641,-24.131,21.555,-43.168
C00759=1016.251,-22.902,382.614,-24.131,21.556,-43.162
C00760=1016.250,-22.569,382.588,-24.132,21.554,-43.158
C00761=1016.249,-22.237,382.562,-24.133,21.554,-43.153
C00762=1016.248,-21.905,382.535,-24.133,21.554,-43.149
C00763=1016.247,-21.572,382.508,-24.134,21.553,-43.144
C00764=1016.246,-21.239,382.483,-24.134,21.552,-43.140
C00765=1016.245,-20.906,382.456,-24.135,21.553,-43.135
C00766=1016.244,-20.573,382.430,-24.136,21.552,-43.131
C00767=1016.243,-20.241,382.403,-24.136,21.551,-43.127
C00768=1016.241,-19.907,382.377,-24.137,21.551,-43.122
C00769=1016.241,-19.735,382.363,-24.137,21.550,-43.118
C00770=1016.240,-19.319,382.330,-24.138,21.550,-43.112
C00771=1016.238,-19.071,382.310,-24.139,21.550,-43.109
C00772=1016.239,-18.809,382.289,-24.139,21.550,-43.107
C00773=1016.237,-18.547,382.268,-24.139,21.549,-43.105
C00774=1016.236,-18.300,382.248,-24.139,21.548,-43.103
C00775=1016.235,-18.079,382.231,-24.140,21.549,-43.100
C00776=1016.234,-17.713,382.202,-24.141,21.548,-43.092
C00777=1016.233,-17.380,382.175,-24.141,21.547,-43.088
C00778=1016.232,-17.048,382.148,-24.142,21.547,-43.083
C00779=1016.230,-16.714,382.122,-24.142,21.547,-43.079
C00780=1016.229,-16.381,382.095,-24.143,21.546,-43.074
C00781=1016.228,-16.046,382.068,-24.144,21.546,-43.070
C00782=1016.226,-15.711,382.042,-24.145,21.546,-43.065
C00783=1016.225,-15.375,382.014,-24.145,21.545,-43.061
C00784=1016.224,-15.036,381.987,-24.146,21.544,-43.055
C00785=1016.222,-14.696,381.961,-24.146,21.544,-43.052
C00786=1016.221,-14.355,381.933,-24.147,21.544,-43.046
C00787=1016.219,-14.010,381.905,-24.147,21.543,-43.042
C00788=1016.218,-13.663,381.877,-24.148,21.543,-43.037
C00789=1016.217,-13.315,381.850,-24.149,21.542,-43.033
C00790=1016.215,-12.965,381.821,-24.149,21.542,-43.028
C00791=1016.214,-12.613,381.793,-24.150,21.541,-43.024
C00792=1016.212,-12.259,381.764,-24.151,21.541,-43.019
C00793=1016.210,-11.904,381.736,-24.151,21.540,-43.014
C00794=1016.208,-11.548,381.707,-24.152,21.540,-43.009
C00795=1016.207,-11.191,381.679,-24.152,21.539,-43.006
C00796=1016.205,-10.832,381.650,-24.153,21.539,-43.000
C00797=1016.203,-10.472,381.620,-24.154,21.539,-42.995
C00798=1016.202,-10.111,381.592,-24.154,21.538,-42.991
C00799=1016.200,-9.750,381.563,-24.155,21.538,-42.985
C00800=1016.198,-9.387,381.533,-24.156,21.537,-42.982
C00801=1016.197,-9.025,381.504,-24.156,21.536,-42.976
C00802=1016.195,-8.663,381.475,-24.157,21.536,-42.971
C00803=1016.193,-8.300,381.445,-24.158,21.536,-42.967
C00804=1016.192,-7.936,381.416,-24.158,21.535,-42.961
C00805=1016.189,-7.570,381.386,-24.159,21.535,-42.956
C00806=1016.187,-7.201,381.357,-24.160,21.534,-42.952
C00807=1016.186,-6.829,381.327,-24.160,21.534,-42.947
C00808=1016.183,-6.455,381.296,-24.161,21.533,-42.941
C00809=1016.182,-6.079,381.266,-24.162,21.533,-42.937
C00810=1016.180,-5.704,381.235,-24.163,21.533,-42.932
C00811=1016.177,-5.331,381.205,-24.163,21.532,-42.928
C00812=1016.176,-4.960,381.175,-24.164,21.532,-42.923
C00813=1016.173,-4.594,381.145,-24.164,21.531,-42.919
C00814=1016.171,-4.232,381.116,-24.165,21.530,-42.913
C00815=1016.170,-3.874,381.088,-24.166,21.531,-42.908
C00816=1016.167,-3.521,381.058,-24.166,21.529,-42.904
C00817=1016.166,-3.168,381.029,-24.167,21.529,-42.899
C00818=1016.164,-2.816,381.001,-24.167,21.529,-42.895
C00819=1016.161,-2.467,380.973,-24.168,21.529,-42.890
C00820=1016.159,-2.118,380.945,-24.169,21.528,-42.886
C00821=1016.157,-1.772,380.916,-24.169,21.528,-42.880
C00822=1016.156,-1.426,380.888,-24.170,21.527,-42.877
C00823=1016.153,-1.083,380.860,-24.170,21.527,-42.873
C00824=1016.151,-0.742,380.832,-24.171,21.526,-42.867
C00825=1016.149,-0.402,380.805,-24.172,21.526,-42.864
C00826=1016.147,-0.063,380.777,-24.172,21.526,-42.858
C00827=1016.145,0.274,380.750,-24.173,21.525,-42.855
C00828=1016.143,0.610,380.722,-24.173,21.525,-42.851
C00829=1016.141,0.945,380.695,-24.174,21.525,-42.846
C00830=1016.138,1.279,380.668,-24.175,21.524,-42.842
C00831=1016.136,1.612,380.640,-24.175,21.523,-42.838
C00832=1016.134,1.943,380.613,-24.176,21.523,-42.834
C00833=1016.132,2.255,380.587,-24.176,21.523,-42.831
C00834=1016.130,2.543,380.564,-24.177,21.522,-42.827
C00835=1016.128,2.812,380.542,-24.177,21.522,-42.823
C00836=1016.127,3.074,380.521,-24.178,21.522,-42.818
C00837=1016.125,3.343,380.499,-24.179,21.521,-42.814
C00838=1016.123,3.633,380.475,-24.179,21.521,-42.810
C00839=1016.121,3.946,380.450,-24.179,21.520,-42.807
C00840=1016.118,4.276,380.422,-24.180,21.521,-42.803
C00841=1016.117,4.607,380.395,-24.180,21.519,-42.799
C00842=1016.114,4.938,380.368,-24.181,21.519,-42.795
C00843=1016.112,5.269,380.341,-24.181,21.518,-42.792
C00844=1016.110,5.599,380.313,-24.182,21.519,-42.786
C00845=1016.107,5.929,380.287,-24.183,21.518,-42.783
C00846=1016.105,6.259,380.260,-24.183,21.518,-42.779
C00847=1016.102,6.588,380.232,-24.184,21.518,-42.774
C00848=1016.100,6.916,380.205,-24.185,21.517,-42.770
C00849=1016.098,7.243,380.179,-24.185,21.517,-42.766
C00850=1016.095,7.569,380.152,-24.186,21.516,-42.762
C00851=1016.094,7.892,380.125,-24.186,21.516,-42.759
C00852=1016.091,8.212,380.099,-24.186,21.515,-42.755
C00853=1016.088,8.531,380.072,-24.187,21.516,-42.750
C00854=1016.086,8.847,380.047,-24.188,21.515,-42.746
C00855=1016.083,9.163,380.021,-24.188,21.515,-42.742
C00856=1016.082,9.477,379.994,-24.189,21.514,-42.738
C00857=1016.079,9.792,379.969,-24.190,21.514,-42.733
C00858=1016.076,10.108,379.942,-24.190,21.514,-42.730
C00859=1016.074,10.424,379.917,-24.191,21.513,-42.726
C00860=1016.071,10.743,379.890,-24.191,21.513,-42.722
C00861=1016.069,11.064,379.864,-24.192,21.512,-42.718
C00862=1016.067,11.386,379.838,-24.192,21.512,-42.715
C00863=1016.065,11.709,379.810,-24.193,21.511,-42.711
C00864=1016.061,12.033,379.784,-24.193,21.511,-42.707
C00865=1016.059,12.357,379.757,-24.194,21.511,-42.702
C00866=1016.056,12.679,379.730,-24.194,21.510,-42.698
C00867=1016.054,13.003,379.703,-24.195,21.510,-42.694
C00868=1016.051,13.327,379.677,-24.195,21.509,-42.691
C00869=1016.048,13.651,379.650,-24.196,21.509,-42.687
C00870=1016.045,13.975,379.623,-24.197,21.509,-42.682
C00871=1016.043,14.300,379.596,-24.197,21.509,-42.678
C00872=1016.040,14.625,379.569,-24.198,21.508,-42.674
C00873=1016.037,14.950,379.542,-24.198,21.508,-42.670
C00874=1016.035,15.277,379.514,-24.199,21.507,-42.667
C00875=1016.032,15.603,379.488,-24.199,21.507,-42.663
C00876=1016.030,15.929,379.461,-24.200,21.507,-42.658
C00877=1016.027,16.258,379.433,-24.200,21.506,-42.654
C00878=1016.023,16.586,379.407,-24.201,21.506,-42.650
C00879=1016.021,16.914,379.379,-24.201,21.505,-42.646
C00880=1016.018,17.243,379.352,-24.202,21.505,-42.643
C00881=1016.015,17.573,379.324,-24.202,21.504,-42.639
C00882=1016.012,17.904,379.297,-24.203,21.504,-42.634
C00883=1016.010,18.233,379.270,-24.204,21.504,-42.630
C00884=1016.006,18.566,379.242,-24.204,21.503,-42.626
C00885=1016.004,18.897,379.215,-24.205,21.503,-42.622
C00886=1016.000,19.229,379.186,-24.205,21.502,-42.619
C00887=1015.997,19.577,379.158,-24.206,21.503,-42.613
C00888=1015.994,19.995,379.123,-24.207,21.502,-42.608
C00889=1015.992,20.231,379.103,-24.207,21.502,-42.604
C00890=1015.989,20.477,379.083,-24.207,21.502,-42.603
C00891=1015.987,20.725,379.062,-24.208,21.502,-42.601
C00892=1015.985,20.967,379.042,-24.208,21.502,-42.599
C00893=1015.982,21.195,379.023,-24.208,21.501,-42.597
C00894=1015.980,21.401,379.006,-24.209,21.501,-42.593
C00895=1015.977,21.759,378.976,-24.209,21.500,-42.588
C00896=1015.975,22.082,378.949,-24.210,21.501,-42.584
C00897=1015.972,22.377,378.924,-24.210,21.500,-42.582
C00898=1015.969,22.630,378.903,-24.210,21.499,-42.580
C00899=1015.966,23.039,378.869,-24.211,21.499,-42.573
C00900=1015.962,23.446,378.835,-24.212,21.498,-42.565
C00901=1015.959,23.699,378.814,-24.213,21.498,-42.562
C00902=1015.956,23.993,378.789,-24.213,21.498,-42.560
C00903=1015.953,24.320,378.762,-24.213,21.497,-42.558
C00904=1015.950,24.654,378.734,-24.214,21.497,-42.553
C00905=1015.947,24.989,378.706,-24.215,21.497,-42.549
C00906=1015.943,25.323,378.679,-24.215,21.496,-42.545
C00907=1015.940,25.657,378.650,-24.216,21.496,-42.541
C00908=1015.936,25.991,378.622,-24.216,21.495,-42.538
C00909=1015.933,26.325,378.595,-24.217,21.495,-42.534
C00910=1015.929,26.660,378.567,-24.217,21.494,-42.530
C00911=1015.927,26.994,378.538,-24.218,21.494,-42.525
C00912=1015.923,27.328,378.510,-24.219,21.495,-42.522
C00913=1015.920,27.663,378.482,-24.219,21.494,-42.518
C00914=1015.916,27.997,378.454,-24.220,21.494,-42.514
C00915=1015.913,28.332,378.426,-24.220,21.493,-42.510
C00916=1015.909,28.666,378.397,-24.221,21.493,-42.507
C00917=1015.906,29.000,378.369,-24.221,21.492,-42.503
C00918=1015.902,29.335,378.341,-24.222,21.493,-42.498
C00919=1015.899,29.669,378.314,-24.222,21.492,-42.494
C00920=1015.896,30.004,378.286,-24.223,21.492,-42.490
C00921=1015.892,30.338,378.258,-24.223,21.491,-42.486
C00922=1015.888,30.672,378.229,-24.224,21.491,-42.483
C00923=1015.885,31.006,378.201,-24.224,21.490,-42.479
C00924=1015.881,31.342,378.173,-24.225,21.490,-42.475
C00925=1015.878,31.676,378.145,-24.225,21.489,-42.471
C00926=1015.874,32.010,378.117,-24.226,21.489,-42.468
C00927=1015.869,32.345,378.089,-24.226,21.489,-42.464
C00928=1015.866,32.680,378.060,-24.227,21.489,-42.459
C00929=1015.862,33.015,378.032,-24.228,21.489,-42.455
C00930=1015.859,33.348,378.004,-24.228,21.488,-42.452
C00931=1015.855,33.683,377.976,-24.229,21.488,-42.448
C00932=1015.852,34.018,377.947,-24.229,21.487,-42.444
C00933=1015.848,34.352,377.919,-24.230,21.487,-42.440
C00934=1015.844,34.687,377.891,-24.230,21.486,-42.437
C00935=1015.840,35.021,377.863,-24.231,21.486,-42.433
C00936=1015.836,35.356,377.835,-24.231,21.485,-42.429
C00937=1015.832,35.691,377.806,-24.232,21.486,-42.426
C00938=1015.828,36.026,377.778,-24.232,21.485,-42.422
C00939=1015.825,36.360,377.750,-24.233,21.485,-42.418
C00940=1015.820,36.695,377.722,-24.234,21.485,-42.413
C00941=1015.817,37.030,377.693,-24.234,21.485,-42.409
C00942=1015.813,37.364,377.665,-24.235,21.484,-42.405
C00943=1015.809,37.699,377.637,-24.235,21.484,-42.402
C00944=1015.805,38.033,377.609,-24.236,21.483,-42.398
C00945=1015.801,38.369,377.580,-24.236,21.483,-42.395
C00946=1015.797,38.703,377.552,-24.237,21.483,-42.391
C00947=1015.793,39.038,377.523,-24.237,21.483,-42.387
C00948=1015.789,39.372,377.495,-24.238,21.482,-42.383
C00949=1015.785,39.708,377.467,-24.238,21.482,-42.380
C00950=1015.781,40.042,377.439,-24.239,21.481,-42.376
C00951=1015.777,40.377,377.410,-24.239,21.481,-42.372
C00952=1015.773,40.711,377.382,-24.240,21.481,-42.369
C00953=1015.768,41.046,377.354,-24.240,21.481,-42.365
C00954=1015.765,41.381,377.325,-24.241,21.480,-42.361
C00955=1015.761,41.716,377.297,-24.241,21.480,-42.357
C00956=1015.756,42.051,377.268,-24.242,21.479,-42.354
C00957=1015.752,42.385,377.240,-24.242,21.479,-42.350
C00958=1015.748,42.720,377.212,-24.243,21.479,-42.347
C00959=1015.744,43.055,377.183,-24.243,21.479,-42.343
C00960=1015.740,43.390,377.154,-24.244,21.478,-42.339
C00961=1015.735,43.725,377.126,-24.244,21.478,-42.335
C00962=1015.731,44.060,377.098,-24.245,21.477,-42.332
C00963=1015.726,44.394,377.070,-24.245,21.477,-42.328
C00964=1015.723,44.730,377.041,-24.246,21.477,-42.325
C00965=1015.718,45.065,377.012,-24.246,21.477,-42.321
C00966=1015.713,45.399,376.984,-24.247,21.476,-42.317
C00967=1015.709,45.734,376.955,-24.247,21.476,-42.313
C00968=1015.704,46.069,376.927,-24.248,21.475,-42.309
C00969=1015.700,46.403,376.898,-24.248,21.475,-42.306
C00970=1015.696,46.739,376.869,-24.249,21.475,-42.302
C00971=1015.692,47.074,376.841,-24.249,21.475,-42.299
C00972=1015.687,47.409,376.814,-24.250,21.474,-42.295
C00973=1015.682,47.744,376.784,-24.250,21.474,-42.291
C00974=1015.678,48.078,376.756,-24.251,21.473,-42.287
C00975=1015.673,48.413,376.727,-24.251,21.473,-42.284
C00976=1015.669,48.748,376.699,-24.252,21.473,-42.280
C00977=1015.665,49.083,376.670,-24.252,21.473,-42.277
C00978=1015.660,49.418,376.641,-24.253,21.472,-42.273
C00979=1015.655,49.753,376.614,-24.253,21.472,-42.269
C00980=1015.651,50.088,376.585,-24.254,21.472,-42.266
C00981=1015.646,50.423,376.556,-24.254,21.471,-42.262
C00982=1015.642,50.757,376.528,-24.255,21.471,-42.258
C00983=1015.637,51.092,376.499,-24.255,21.471,-42.254
C00984=1015.632,51.427,376.470,-24.256,21.471,-42.251
C00985=1015.627,51.763,376.442,-24.256,21.470,-42.247
C00986=1015.623,52.097,376.414,-24.257,21.470,-42.244
C00987=1015.617,52.432,376.385,-24.257,21.470,-42.240
C00988=1015.613,52.767,376.356,-24.258,21.469,-42.238
C00989=1015.608,53.102,376.328,-24.258,21.469,-42.234
C00990=1015.604,53.436,376.299,-24.259,21.468,-42.230
C00991=1015.598,53.772,376.271,-24.259,21.468,-42.227
C00992=1015.594,54.107,376.242,-24.260,21.468,-42.223
C00993=1015.589,54.442,376.214,-24.260,21.468,-42.220
C00994=1015.584,54.777,376.184,-24.261,21.467,-42.216
C00995=1015.580,55.111,376.156,-24.261,21.467,-42.212
C00996=1015.574,55.447,376.128,-24.262,21.467,-42.209
C00997=1015.570,55.782,376.099,-24.262,21.467,-42.205
C00998=1015.564,56.117,376.070,-24.263,21.466,-42.201
C00999=1015.560,56.451,376.041,-24.263,21.466,-42.197
C01000=1015.555,56.786,376.013,-24.264,21.466,-42.194
C01001=1015.550,57.122,375.984,-24.264,21.465,-42.192
C01002=1015.545,57.457,375.956,-24.264,21.465,-42.188
C01003=1015.540,57.792,375.927,-24.265,21.464,-42.184
C01004=1015.535,58.127,375.898,-24.266,21.465,-42.181
C01005=1015.529,58.461,375.870,-24.266,21.464,-42.177
C01006=1015.524,58.796,375.841,-24.267,21.464,-42.173
C01007=1015.519,59.131,375.812,-24.267,21.464,-42.170
C01008=1015.514,59.466,375.783,-24.268,21.464,-42.166
C01009=1015.509,59.801,375.754,-24.268,21.463,-42.163
C01010=1015.504,60.136,375.726,-24.268,21.462,-42.160
C01011=1015.498,60.471,375.697,-24.269,21.462,-42.157
C01012=1015.493,60.806,375.668,-24.269,21.462,-42.153
C01013=1015.489,61.141,375.640,-24.270,21.461,-42.149
C01014=1015.483,61.476,375.611,-24.270,21.462,-42.146
C01015=1015.477,61.811,375.583,-24.271,21.461,-42.142
C01016=1015.473,62.145,375.554,-24.271,21.461,-42.139
C01017=1015.467,62.482,375.525,-24.272,21.460,-42.135
C01018=1015.461,62.878,375.490,-24.272,21.460,-42.131
C01019=1015.458,63.102,375.472,-24.273,21.461,-42.130
C01020=1015.454,63.320,375.453,-24.273,21.460,-42.128
C01021=1015.449,63.694,375.420,-24.274,21.460,-42.124
C01022=1015.448,64.049,375.386,-24.274,21.459,-42.120
C01023=1015.448,64.436,375.350,-24.274,21.459,-42.116
C01024=1015.446,64.831,375.313,-24.275,21.458,-42.113
C01025=1015.445,65.209,375.278,-24.276,21.459,-42.108
C01026=1015.443,65.562,375.244,-24.276,21.457,-42.105
C01027=1015.443,65.902,375.213,-24.277,21.458,-42.102
C01028=1015.442,66.235,375.181,-24.277,21.457,-42.098
C01029=1015.441,66.570,375.150,-24.278,21.457,-42.094
C01030=1015.440,66.907,375.118,-24.278,21.457,-42.091
C01031=1015.438,67.244,375.086,-24.279,21.457,-42.087
C01032=1015.437,67.582,375.054,-24.279,21.456,-42.085
C01033=1015.437,67.922,375.022,-24.279,21.456,-42.082
C01034=1015.436,68.262,374.990,-24.280,21.456,-42.078
C01035=1015.434,68.603,374.958,-24.280,21.455,-42.074
C01036=1015.433,68.945,374.925,-24.281,21.456,-42.071
C01037=1015.432,69.288,374.892,-24.281,21.455,-42.067
C01038=1015.431,69.632,374.860,-24.282,21.455,-42.063
C01039=1015.430,69.977,374.828,-24.282,21.454,-42.061
C01040=1015.429,70.322,374.795,-24.283,21.454,-42.058
C01041=1015.428,70.666,374.763,-24.283,21.453,-42.054
C01042=1015.427,71.010,374.730,-24.284,21.454,-42.051
C01043=1015.426,71.355,374.697,-24.284,21.453,-42.047
C01044=1015.425,71.699,374.664,-24.285,21.453,-42.043
C01045=1015.423,72.045,374.631,-24.285,21.453,-42.041
C01046=1015.422,72.391,374.598,-24.285,21.452,-42.037
C01047=1015.421,72.739,374.565,-24.286,21.452,-42.034
C01048=1015.420,73.089,374.532,-24.286,21.451,-42.030
C01049=1015.419,73.440,374.499,-24.287,21.452,-42.027
C01050=1015.418,73.793,374.465,-24.288,21.451,-42.023
C01051=1015.417,74.149,374.431,-24.288,21.451,-42.019
C01052=1015.415,74.505,374.398,-24.288,21.451,-42.017
C01053=1015.414,74.864,374.364,-24.289,21.450,-42.013
C01054=1015.413,75.221,374.329,-24.289,21.450,-42.010
C01055=1015.412,75.575,374.295,-24.290,21.450,-42.006
C01056=1015.411,75.923,374.263,-24.290,21.449,-42.004
C01057=1015.409,76.266,374.230,-24.291,21.449,-42.001
C01058=1015.408,76.602,374.198,-24.291,21.449,-41.997
C01059=1015.407,76.932,374.166,-24.292,21.449,-41.994
C01060=1015.406,77.258,374.135,-24.292,21.449,-41.990
C01061=1015.405,77.582,374.105,-24.292,21.448,-41.987
C01062=1015.404,77.905,374.073,-24.293,21.448,-41.984
C01063=1015.403,78.230,374.043,-24.293,21.448,-41.980
C01064=1015.402,78.557,374.011,-24.294,21.447,-41.977
C01065=1015.401,78.891,373.979,-24.295,21.448,-41.973
C01066=1015.399,79.229,373.947,-24.295,21.446,-41.971
C01067=1015.398,79.574,373.914,-24.295,21.447,-41.968
C01068=1015.397,79.926,373.879,-24.296,21.446,-41.964
C01069=1015.396,80.280,373.846,-24.296,21.446,-41.962
C01070=1015.394,80.637,373.812,-24.297,21.446,-41.958
C01071=1015.393,80.995,373.777,-24.297,21.445,-41.955
C01072=1015.393,81.350,373.743,-24.298,21.446,-41.951
C01073=1015.390,81.705,373.709,-24.298,21.445,-41.947
C01074=1015.389,82.059,373.675,-24.298,21.444,-41.945
C01075=1015.389,82.413,373.641,-24.299,21.444,-41.942
C01076=1015.387,82.767,373.607,-24.299,21.444,-41.938
C01077=1015.386,83.118,373.574,-24.300,21.444,-41.935
C01078=1015.385,83.469,373.540,-24.300,21.444,-41.931
C01079=1015.384,83.819,373.506,-24.301,21.443,-41.929
C01080=1015.382,84.168,373.472,-24.301,21.443,-41.925
C01081=1015.381,84.516,373.439,-24.302,21.443,-41.922
C01082=1015.380,84.862,373.406,-24.302,21.443,-41.918
C01083=1015.379,85.208,373.372,-24.302,21.442,-41.916
C01084=1015.377,85.552,373.339,-24.303,21.442,-41.912
C01085=1015.377,85.895,373.306,-24.303,21.442,-41.909
C01086=1015.375,86.237,373.273,-24.304,21.441,-41.906
C01087=1015.374,86.578,373.240,-24.304,21.441,-41.903
C01088=1015.372,86.917,373.207,-24.305,21.441,-41.899
C01089=1015.371,87.254,373.175,-24.305,21.441,-41.898
C01090=1015.370,87.587,373.142,-24.305,21.440,-41.894
C01091=1015.369,87.913,373.111,-24.306,21.441,-41.890
C01092=1015.368,88.235,373.080,-24.306,21.439,-41.888
C01093=1015.366,88.556,373.048,-24.307,21.440,-41.885
C01094=1015.366,88.877,373.018,-24.307,21.439,-41.881
C01095=1015.365,89.201,372.986,-24.308,21.439,-41.879
C01096=1015.363,89.531,372.955,-24.308,21.440,-41.876
C01097=1015.362,89.864,372.921,-24.308,21.438,-41.874
C01098=1015.361,90.198,372.890,-24.309,21.439,-41.870
C01099=1015.360,90.533,372.857,-24.309,21.438,-41.866
C01100=1015.358,90.867,372.825,-24.310,21.438,-41.865
C01101=1015.357,91.201,372.792,-24.310,21.438,-41.861
C01102=1015.356,91.536,372.759,-24.311,21.438,-41.857
C01103=1015.354,91.871,372.727,-24.311,21.437,-41.855
C01104=1015.353,92.205,372.695,-24.311,21.437,-41.852
C01105=1015.352,92.539,372.662,-24.312,21.436,-41.849
C01106=1015.350,92.874,372.630,-24.312,21.437,-41.846
C01107=1015.349,93.208,372.597,-24.313,21.436,-41.842
C01108=1015.348,93.542,372.564,-24.313,21.436,-41.841
C01109=1015.347,93.877,372.531,-24.314,21.436,-41.837
C01110=1015.346,94.211,372.499,-24.314,21.436,-41.833
C01111=1015.345,94.545,372.467,-24.314,21.436,-41.832
C01112=1015.343,94.879,372.434,-24.315,21.435,-41.828
C01113=1015.342,95.214,372.402,-24.315,21.435,-41.826
C01114=1015.340,95.548,372.369,-24.316,21.435,-41.822
C01115=1015.340,95.883,372.336,-24.316,21.435,-41.819
C01116=1015.338,96.217,372.303,-24.316,21.434,-41.817
C01117=1015.337,96.551,372.271,-24.317,21.434,-41.813
C01118=1015.335,96.886,372.238,-24.317,21.434,-41.811
C01119=1015.335,97.219,372.206,-24.318,21.434,-41.808
C01120=1015.333,97.553,372.173,-24.318,21.433,-41.806
C01121=1015.332,97.888,372.141,-24.318,21.433,-41.802
C01122=1015.331,98.221,372.107,-24.319,21.433,-41.799
C01123=1015.329,98.556,372.075,-24.319,21.432,-41.796
C01124=1015.328,98.890,372.042,-24.320,21.433,-41.793
C01125=1015.326,99.224,372.009,-24.320,21.432,-41.791
C01126=1015.326,99.559,371.976,-24.320,21.432,-41.787
C01127=1015.324,99.893,371.944,-24.321,21.432,-41.785
C01128=1015.323,100.227,371.910,-24.321,21.431,-41.782
C01129=1015.321,100.561,371.878,-24.322,21.432,-41.778
C01130=1015.320,100.896,371.845,-24.322,21.431,-41.776
C01131=1015.319,101.229,371.812,-24.323,21.431,-41.773
C01132=1015.317,101.564,371.780,-24.323,21.431,-41.771
C01133=1015.316,101.897,371.747,-24.323,21.430,-41.767
C01134=1015.315,102.232,371.714,-24.324,21.430,-41.765
C01135=1015.313,102.565,371.681,-24.324,21.431,-41.762
C01136=1015.312,102.900,371.648,-24.324,21.429,-41.760
C01137=1015.311,103.234,371.615,-24.325,21.430,-41.756
C01138=1015.309,103.568,371.583,-24.325,21.429,-41.752
C01139=1015.308,103.902,371.549,-24.326,21.429,-41.751
C01140=1015.307,104.236,371.517,-24.326,21.430,-41.747
C01141=1015.305,104.570,371.484,-24.326,21.428,-41.745
C01142=1015.304,104.904,371.451,-24.327,21.429,-41.742
C01143=1015.303,105.238,371.418,-24.327,21.428,-41.739
C01144=1015.302,105.573,371.385,-24.328,21.428,-41.736
C01145=1015.301,105.906,371.352,-24.328,21.428,-41.734
C01146=1015.300,106.240,371.319,-24.328,21.427,-41.730
C01147=1015.298,106.575,371.286,-24.329,21.427,-41.728
C01148=1015.297,106.908,371.253,-24.329,21.428,-41.725
C01149=1015.295,107.243,371.220,-24.329,21.427,-41.723
C01150=1015.293,107.577,371.187,-24.330,21.427,-41.719
C01151=1015.292,107.910,371.153,-24.330,21.427,-41.718
C01152=1015.291,108.245,371.121,-24.331,21.426,-41.714
C01153=1015.290,108.578,371.088,-24.331,21.426,-41.712
C01154=1015.288,108.912,371.054,-24.332,21.426,-41.708
C01155=1015.287,109.246,371.022,-24.332,21.425,-41.706
C01156=1015.286,109.580,370.989,-24.332,21.426,-41.703
C01157=1015.285,109.914,370.955,-24.333,21.425,-41.701
C01158=1015.283,110.248,370.922,-24.333,21.425,-41.697
C01159=1015.281,110.582,370.889,-24.333,21.425,-41.695
C01160=1015.280,110.916,370.856,-24.334,21.424,-41.692
C01161=1015.279,111.250,370.823,-24.334,21.424,-41.690
C01162=1015.278,111.583,370.789,-24.335,21.425,-41.686
C01163=1015.276,111.918,370.757,-24.335,21.423,-41.684
C01164=1015.274,112.252,370.723,-24.335,21.424,-41.681
C01165=1015.273,112.586,370.690,-24.336,21.424,-41.679
C01166=1015.272,112.919,370.657,-24.336,21.423,-41.675
C01167=1015.270,113.254,370.624,-24.336,21.423,-41.673
C01168=1015.269,113.588,370.590,-24.337,21.423,-41.670
C01169=1015.268,113.922,370.557,-24.337,21.422,-41.668
C01170=1015.267,114.256,370.524,-24.338,21.423,-41.664
C01171=1015.266,114.590,370.490,-24.338,21.422,-41.662
C01172=1015.264,114.923,370.457,-24.338,21.421,-41.660
C01173=1015.262,115.258,370.424,-24.339,21.422,-41.657
C01174=1015.261,115.592,370.391,-24.339,21.422,-41.655
C01175=1015.260,115.925,370.358,-24.340,21.422,-41.652
C01176=1015.258,116.259,370.324,-24.340,21.421,-41.649
C01177=1015.257,116.593,370.291,-24.340,21.421,-41.646
C01178=1015.256,116.927,370.257,-24.341,21.421,-41.644
C01179=1015.254,117.261,370.224,-24.341,21.421,-41.640
C01180=1015.252,117.595,370.190,-24.341,21.420,-41.638
C01181=1015.252,117.929,370.157,-24.342,21.421,-41.635
C01182=1015.251,118.263,370.124,-24.342,21.420,-41.633
C01183=1015.248,118.597,370.090,-24.342,21.419,-41.631
C01184=1015.247,118.931,370.057,-24.343,21.420,-41.628
C01185=1015.245,119.265,370.023,-24.343,21.419,-41.625
C01186=1015.244,119.599,369.990,-24.344,21.419,-41.622
C01187=1015.243,119.933,369.957,-24.344,21.419,-41.620
C01188=1015.241,120.267,369.923,-24.345,21.419,-41.617
C01189=1015.240,120.600,369.890,-24.345,21.418,-41.614
C01190=1015.239,120.935,369.856,-24.345,21.418,-41.613
C01191=1015.237,121.269,369.823,-24.346,21.418,-41.609
C01192=1015.236,121.603,369.789,-24.346,21.417,-41.607
C01193=1015.234,121.937,369.755,-24.346,21.418,-41.604
C01194=1015.233,122.270,369.722,-24.347,21.418,-41.602
C01195=1015.232,122.604,369.689,-24.347,21.418,-41.598
C01196=1015.230,122.938,369.655,-24.347,21.417,-41.596
C01197=1015.229,123.272,369.622,-24.348,21.417,-41.594
C01198=1015.228,123.606,369.588,-24.348,21.417,-41.591
C01199=1015.226,123.940,369.555,-24.348,21.417,-41.589
C01200=1015.225,124.274,369.520,-24.349,21.416,-41.585
C01201=1015.224,124.607,369.487,-24.349,21.416,-41.583
C01202=1015.222,124.942,369.453,-24.349,21.416,-41.581
C01203=1015.221,125.276,369.419,-24.350,21.416,-41.578
C01204=1015.219,125.610,369.386,-24.350,21.415,-41.576
C01205=1015.218,125.944,369.352,-24.351,21.416,-41.572
C01206=1015.216,126.278,369.319,-24.351,21.415,-41.571
C01207=1015.215,126.612,369.285,-24.351,21.415,-41.569
C01208=1015.214,126.946,369.251,-24.352,21.415,-41.565
C01209=1015.212,127.280,369.218,-24.352,21.415,-41.563
C01210=1015.210,127.614,369.184,-24.352,21.414,-41.561
C01211=1015.209,127.948,369.149,-24.353,21.415,-41.558
C01212=1015.208,128.282,369.116,-24.353,21.414,-41.555
C01213=1015.206,128.616,369.082,-24.354,21.414,-41.552
C01214=1015.205,128.949,369.049,-24.354,21.414,-41.550
C01215=1015.204,129.284,369.015,-24.354,21.414,-41.548
C01216=1015.202,129.618,368.981,-24.355,21.413,-41.545
C01217=1015.201,129.952,368.948,-24.355,21.413,-41.543
C01218=1015.200,130.286,368.913,-24.355,21.413,-41.541
C01219=1015.198,130.620,368.879,-24.356,21.413,-41.538
C01220=1015.197,130.954,368.846,-24.356,21.412,-41.535
C01221=1015.195,131.288,368.812,-24.356,21.412,-41.532
C01222=1015.193,131.623,368.778,-24.357,21.412,-41.530
C01223=1015.192,131.956,368.745,-24.357,21.412,-41.528
C01224=1015.191,132.290,368.710,-24.357,21.412,-41.525
C01225=1015.189,132.624,368.676,-24.358,21.411,-41.523
C01226=1015.189,132.959,368.642,-24.358,21.411,-41.521
C01227=1015.187,133.293,368.609,-24.358,21.411,-41.517
C01228=1015.185,133.627,368.575,-24.359,21.411,-41.515
C01229=1015.184,133.961,368.540,-24.359,21.410,-41.513
C01230=1015.183,134.295,368.507,-24.359,21.411,-41.510
C01231=1015.181,134.629,368.472,-24.360,21.410,-41.508
C01232=1015.179,134.964,368.439,-24.360,21.410,-41.506
C01233=1015.179,135.297,368.405,-24.361,21.411,-41.503
C01234=1015.177,135.620,368.372,-24.361,21.410,-41.501
C01235=1015.175,135.920,368.341,-24.361,21.410,-41.499
C01236=1015.174,136.200,368.313,-24.361,21.410,-41.497
C01237=1015.174,136.464,368.286,-24.361,21.409,-41.495
C01238=1015.172,136.729,368.258,-24.362,21.409,-41.491
C01239=1015.171,137.005,368.231,-24.362,21.409,-41.490
C01240=1015.170,137.302,368.201,-24.363,21.409,-41.488
C01241=1015.168,137.625,368.167,-24.363,21.408,-41.486
C01242=1015.167,137.965,368.132,-24.363,21.408,-41.484
C01243=1015.166,138.321,368.096,-24.364,21.408,-41.480
C01244=1015.164,138.732,368.055,-24.364,21.408,-41.477
C01245=1015.163,138.960,368.031,-24.364,21.408,-41.475
C01246=1015.162,139.198,368.006,-24.365,21.408,-41.473
C01247=1015.160,139.440,367.982,-24.365,21.408,-41.473
C01248=1015.160,139.681,367.958,-24.365,21.408,-41.471
C01249=1015.159,139.914,367.933,-24.365,21.408,-41.470
C01250=1015.159,140.134,367.911,-24.365,21.407,-41.469
C01251=1015.156,140.527,367.871,-24.366,21.407,-41.465
C01252=1015.155,140.873,367.835,-24.366,21.407,-41.462
C01253=1015.154,141.211,367.801,-24.367,21.407,-41.460
C01254=1015.153,141.551,367.766,-24.367,21.407,-41.457
C01255=1015.151,141.891,367.730,-24.367,21.406,-41.455
C01256=1015.149,142.232,367.696,-24.368,21.406,-41.453
C01257=1015.147,142.573,367.661,-24.368,21.407,-41.449
C01258=1015.146,142.915,367.625,-24.368,21.406,-41.448
C01259=1015.145,143.257,367.590,-24.369,21.405,-41.445
C01260=1015.144,143.601,367.555,-24.369,21.406,-41.442
C01261=1015.141,143.944,367.520,-24.369,21.405,-41.440
C01262=1015.141,144.288,367.485,-24.370,21.405,-41.438
C01263=1015.140,144.633,367.449,-24.370,21.406,-41.435
C01264=1015.138,144.978,367.415,-24.370,21.405,-41.432
C01265=1015.136,145.323,367.378,-24.371,21.404,-41.431
C01266=1015.135,145.669,367.342,-24.371,21.405,-41.427
C01267=1015.134,146.014,367.307,-24.371,21.405,-41.425
C01268=1015.132,146.362,367.272,-24.372,21.404,-41.424
C01269=1015.130,146.707,367.236,-24.372,21.404,-41.420
C01270=1015.122,147.053,367.204,-24.372,21.404,-41.418
C01271=1015.538,147.083,366.945,-24.372,21.404,-41.418
C01272=1015.549,146.738,366.976,-24.372,21.404,-41.420
C01273=1015.550,146.391,367.011,-24.372,21.404,-41.424
C01274=1015.552,146.045,367.046,-24.371,21.405,-41.425
C01275=1015.553,145.699,367.082,-24.371,21.405,-41.427
C01276=1015.555,145.353,367.118,-24.371,21.404,-41.431
C01277=1015.556,145.008,367.154,-24.370,21.405,-41.432
C01278=1015.557,144.663,367.189,-24.370,21.406,-41.435
C01279=1015.559,144.319,367.224,-24.370,21.405,-41.438
C01280=1015.560,143.975,367.260,-24.369,21.405,-41.440
C01281=1015.561,143.631,367.295,-24.369,21.406,-41.442
C01282=1015.563,143.287,367.330,-24.369,21.405,-41.445
C01283=1015.564,142.945,367.365,-24.368,21.406,-41.448
C01284=1015.566,142.603,367.400,-24.368,21.407,-41.449
C01285=1015.567,142.262,367.435,-24.368,21.406,-41.453
C01286=1015.569,141.921,367.470,-24.367,21.406,-41.455
C01287=1015.570,141.581,367.505,-24.367,21.407,-41.457
C01288=1015.572,141.242,367.540,-24.367,21.407,-41.460
C01289=1015.573,140.902,367.575,-24.366,21.407,-41.462
C01290=1015.575,140.558,367.610,-24.366,21.407,-41.465
C01291=1015.576,140.164,367.650,-24.365,21.407,-41.469
C01292=1015.577,139.943,367.673,-24.365,21.408,-41.470
C01293=1015.577,139.711,367.697,-24.365,21.408,-41.471
C01294=1015.578,139.470,367.721,-24.365,21.408,-41.473
C01295=1015.579,139.229,367.746,-24.365,21.408,-41.473
C01296=1015.581,138.990,367.770,-24.364,21.408,-41.475
C01297=1015.582,138.763,367.794,-24.364,21.408,-41.477
C01298=1015.583,138.351,367.836,-24.364,21.408,-41.480
C01299=1015.584,137.995,367.872,-24.363,21.408,-41.484
C01300=1015.586,137.654,367.907,-24.363,21.408,-41.486
C01301=1015.587,137.332,367.940,-24.363,21.409,-41.488
C01302=1015.589,137.035,367.971,-24.362,21.409,-41.490
C01303=1015.589,136.759,367.998,-24.362,21.409,-41.491
C01304=1015.591,136.495,368.026,-24.361,21.409,-41.495
C01305=1015.592,136.230,368.052,-24.361,21.410,-41.497
C01306=1015.593,135.950,368.081,-24.361,21.410,-41.499
C01307=1015.594,135.650,368.111,-24.361,21.410,-41.501
C01308=1015.596,135.327,368.145,-24.361,21.411,-41.503
C01309=1015.597,134.994,368.178,-24.360,21.410,-41.506
C01310=1015.599,134.659,368.212,-24.360,21.410,-41.508
C01311=1015.600,134.325,368.247,-24.359,21.411,-41.510
C01312=1015.602,133.991,368.281,-24.359,21.410,-41.513
C01313=1015.602,133.657,368.314,-24.359,21.411,-41.515
C01314=1015.604,133.323,368.348,-24.358,21.411,-41.517
C01315=1015.605,132.989,368.383,-24.358,21.411,-41.521
C01316=1015.606,132.655,368.416,-24.358,21.411,-41.523
C01317=1015.608,132.321,368.450,-24.357,21.412,-41.525
C01318=1015.610,131.986,368.484,-24.357,21.412,-41.528
C01319=1015.612,131.652,368.518,-24.357,21.412,-41.530
C01320=1015.612,131.319,368.552,-24.356,21.412,-41.532
C01321=1015.614,130.984,368.586,-24.356,21.412,-41.535
C01322=1015.616,130.650,368.620,-24.356,21.413,-41.538
C01323=1015.616,130.316,368.653,-24.355,21.413,-41.541
C01324=1015.618,129.982,368.687,-24.355,21.413,-41.543
C01325=1015.619,129.649,368.721,-24.355,21.413,-41.545
C01326=1015.620,129.314,368.755,-24.354,21.414,-41.548
C01327=1015.622,128.980,368.789,-24.354,21.414,-41.550
C01328=1015.623,128.646,368.822,-24.354,21.414,-41.552
C01329=1015.625,128.312,368.856,-24.353,21.414,-41.555
C01330=1015.626,127.978,368.890,-24.353,21.415,-41.558
C01331=1015.628,127.644,368.924,-24.352,21.414,-41.561
C01332=1015.629,127.310,368.958,-24.352,21.415,-41.563
C01333=1015.630,126.976,368.992,-24.352,21.415,-41.565
C01334=1015.632,126.642,369.025,-24.351,21.415,-41.569
C01335=1015.633,126.308,369.059,-24.351,21.415,-41.571
C01336=1015.634,125.973,369.093,-24.351,21.416,-41.572
C01337=1015.636,125.640,369.126,-24.350,21.415,-41.576
C01338=1015.638,125.306,369.160,-24.350,21.416,-41.578
C01339=1015.639,124.972,369.193,-24.349,21.416,-41.581
C01340=1015.641,124.638,369.227,-24.349,21.416,-41.583
C01341=1015.641,124.304,369.261,-24.349,21.416,-41.585
C01342=1015.643,123.970,369.295,-24.348,21.417,-41.589
C01343=1015.644,123.636,369.328,-24.348,21.417,-41.591
C01344=1015.645,123.303,369.361,-24.348,21.417,-41.594
C01345=1015.647,122.969,369.395,-24.347,21.417,-41.596
C01346=1015.648,122.634,369.429,-24.347,21.418,-41.598
C01347=1015.650,122.300,369.463,-24.347,21.418,-41.602
C01348=1015.651,121.966,369.496,-24.346,21.418,-41.604
C01349=1015.653,121.632,369.530,-24.346,21.417,-41.607
C01350=1015.654,121.299,369.563,-24.346,21.418,-41.609
C01351=1015.655,120.965,369.596,-24.345,21.418,-41.613
C01352=1015.656,120.630,369.630,-24.345,21.418,-41.614
C01353=1015.658,120.297,369.664,-24.345,21.419,-41.617
C01354=1015.659,119.962,369.697,-24.344,21.419,-41.620
C01355=1015.661,119.629,369.731,-24.344,21.419,-41.622
C01356=1015.662,119.295,369.764,-24.343,21.419,-41.625
C01357=1015.664,118.961,369.798,-24.343,21.420,-41.628
C01358=1015.665,118.627,369.831,-24.342,21.419,-41.631
C01359=1015.665,118.293,369.864,-24.342,21.420,-41.633
C01360=1015.667,117.959,369.898,-24.342,21.421,-41.635
C01361=1015.669,117.625,369.931,-24.341,21.420,-41.638
C01362=1015.670,117.291,369.965,-24.341,21.421,-41.640
C01363=1015.672,116.957,369.999,-24.341,21.421,-41.644
C01364=1015.673,116.623,370.031,-24.340,21.421,-41.646
C01365=1015.674,116.289,370.064,-24.340,21.421,-41.649
C01366=1015.676,115.956,370.097,-24.340,21.422,-41.652
C01367=1015.677,115.622,370.131,-24.339,21.422,-41.655
C01368=1015.678,115.287,370.165,-24.339,21.422,-41.657
C01369=1015.679,114.953,370.198,-24.338,21.421,-41.660
C01370=1015.680,114.620,370.231,-24.338,21.422,-41.662
C01371=1015.682,114.286,370.265,-24.338,21.423,-41.664
C01372=1015.684,113.951,370.298,-24.337,21.422,-41.668
C01373=1015.685,113.618,370.331,-24.337,21.423,-41.670
C01374=1015.686,113.284,370.364,-24.336,21.423,-41.673
C01375=1015.687,112.950,370.397,-24.336,21.423,-41.675
C01376=1015.689,112.616,370.431,-24.336,21.424,-41.679
C01377=1015.690,112.282,370.464,-24.335,21.424,-41.681
C01378=1015.692,111.948,370.497,-24.335,21.423,-41.684
C01379=1015.693,111.614,370.530,-24.335,21.425,-41.686
C01380=1015.694,111.281,370.563,-24.334,21.424,-41.690
C01381=1015.696,110.946,370.597,-24.334,21.424,-41.692
C01382=1015.697,110.612,370.630,-24.333,21.425,-41.695
C01383=1015.698,110.278,370.663,-24.333,21.425,-41.697
C01384=1015.699,109.944,370.696,-24.333,21.425,-41.701
C01385=1015.701,109.610,370.730,-24.332,21.426,-41.703
C01386=1015.702,109.276,370.762,-24.332,21.425,-41.706
C01387=1015.703,108.942,370.795,-24.332,21.426,-41.708
C01388=1015.705,108.608,370.829,-24.331,21.426,-41.712
C01389=1015.707,108.274,370.862,-24.331,21.426,-41.714
C01390=1015.708,107.940,370.895,-24.330,21.427,-41.718
C01391=1015.709,107.606,370.928,-24.330,21.427,-41.719
C01392=1015.710,107.272,370.961,-24.329,21.427,-41.723
C01393=1015.712,106.938,370.994,-24.329,21.428,-41.725
C01394=1015.713,106.605,371.027,-24.329,21.427,-41.728
C01395=1015.714,106.270,371.060,-24.328,21.427,-41.730
C01396=1015.716,105.937,371.093,-24.328,21.428,-41.734
C01397=1015.717,105.603,371.126,-24.328,21.428,-41.736
C01398=1015.718,105.268,371.159,-24.327,21.428,-41.739
C01399=1015.719,104.934,371.192,-24.327,21.429,-41.742
C01400=1015.720,104.600,371.225,-24.326,21.428,-41.745
C01401=1015.721,104.266,371.258,-24.326,21.430,-41.747
C01402=1015.723,103.932,371.290,-24.326,21.429,-41.751
C01403=1015.724,103.598,371.323,-24.325,21.429,-41.752
C01404=1015.726,103.264,371.356,-24.325,21.430,-41.756
C01405=1015.727,102.930,371.389,-24.324,21.429,-41.760
C01406=1015.728,102.596,371.422,-24.324,21.431,-41.762
C01407=1015.729,102.262,371.455,-24.324,21.430,-41.765
C01408=1015.731,101.928,371.487,-24.323,21.430,-41.767
C01409=1015.732,101.594,371.521,-24.323,21.431,-41.771
C01410=1015.734,101.259,371.553,-24.323,21.431,-41.773
C01411=1015.735,100.926,371.586,-24.322,21.431,-41.776
C01412=1015.736,100.591,371.619,-24.322,21.432,-41.778
C01413=1015.737,100.257,371.652,-24.321,21.431,-41.782
C01414=1015.738,99.923,371.685,-24.321,21.432,-41.785
C01415=1015.740,99.588,371.717,-24.320,21.432,-41.787
C01416=1015.741,99.255,371.751,-24.320,21.432,-41.791
C01417=1015.742,98.920,371.783,-24.320,21.433,-41.793
C01418=1015.744,98.586,371.816,-24.319,21.432,-41.796
C01419=1015.745,98.252,371.849,-24.319,21.433,-41.799
C01420=1015.747,97.918,371.881,-24.318,21.433,-41.802
C01421=1015.748,97.583,371.914,-24.318,21.433,-41.806
C01422=1015.749,97.250,371.947,-24.318,21.434,-41.808
C01423=1015.750,96.915,371.980,-24.317,21.434,-41.811
C01424=1015.752,96.580,372.013,-24.317,21.434,-41.813
C01425=1015.752,96.247,372.045,-24.316,21.434,-41.817
C01426=1015.754,95.913,372.078,-24.316,21.435,-41.819
C01427=1015.755,95.578,372.110,-24.316,21.435,-41.822
C01428=1015.757,95.244,372.143,-24.315,21.435,-41.826
C01429=1015.758,94.910,372.175,-24.315,21.435,-41.828
C01430=1015.759,94.575,372.209,-24.314,21.436,-41.832
C01431=1015.760,94.241,372.241,-24.314,21.436,-41.833
C01432=1015.762,93.906,372.274,-24.314,21.436,-41.837
C01433=1015.762,93.572,372.306,-24.313,21.436,-41.841
C01434=1015.764,93.238,372.338,-24.313,21.436,-41.842
C01435=1015.765,92.904,372.371,-24.312,21.437,-41.846
C01436=1015.766,92.569,372.404,-24.312,21.436,-41.849
C01437=1015.767,92.235,372.437,-24.311,21.437,-41.852
C01438=1015.769,91.901,372.469,-24.311,21.437,-41.855
C01439=1015.770,91.567,372.501,-24.311,21.438,-41.857
C01440=1015.771,91.232,372.534,-24.310,21.438,-41.861
C01441=1015.772,90.897,372.567,-24.310,21.438,-41.865
C01442=1015.773,90.563,372.599,-24.309,21.438,-41.866
C01443=1015.775,90.228,372.632,-24.309,21.439,-41.870
C01444=1015.776,89.894,372.663,-24.308,21.438,-41.874
C01445=1015.777,89.560,372.696,-24.308,21.440,-41.876
C01446=1015.779,89.231,372.728,-24.308,21.439,-41.879
C01447=1015.780,88.907,372.760,-24.307,21.439,-41.881
C01448=1015.780,88.586,372.790,-24.307,21.440,-41.885
C01449=1015.782,88.265,372.822,-24.306,21.439,-41.888
C01450=1015.783,87.943,372.853,-24.306,21.441,-41.890
C01451=1015.784,87.617,372.884,-24.305,21.440,-41.894
C01452=1015.785,87.284,372.917,-24.305,21.441,-41.898
C01453=1015.786,86.948,372.949,-24.305,21.441,-41.899
C01454=1015.787,86.608,372.982,-24.304,21.441,-41.903
C01455=1015.789,86.267,373.015,-24.304,21.441,-41.906
C01456=1015.791,85.925,373.048,-24.303,21.442,-41.909
C01457=1015.791,85.582,373.081,-24.303,21.442,-41.912
C01458=1015.793,85.238,373.114,-24.302,21.442,-41.916
C01459=1015.794,84.892,373.148,-24.302,21.443,-41.918
C01460=1015.795,84.546,373.181,-24.302,21.443,-41.922
C01461=1015.796,84.198,373.214,-24.301,21.443,-41.925
C01462=1015.797,83.849,373.248,-24.301,21.443,-41.929
C01463=1015.799,83.499,373.282,-24.300,21.444,-41.931
C01464=1015.800,83.148,373.316,-24.300,21.444,-41.935
C01465=1015.801,82.796,373.350,-24.299,21.444,-41.938
C01466=1015.802,82.444,373.383,-24.299,21.444,-41.942
C01467=1015.803,82.089,373.417,-24.298,21.444,-41.945
C01468=1015.804,81.735,373.451,-24.298,21.445,-41.947
C01469=1015.806,81.379,373.486,-24.298,21.446,-41.951
C01470=1015.807,81.024,373.520,-24.297,21.445,-41.955
C01471=1015.808,80.668,373.554,-24.297,21.446,-41.958
C01472=1015.810,80.310,373.588,-24.296,21.446,-41.962
C01473=1015.810,79.956,373.622,-24.296,21.446,-41.964
C01474=1015.812,79.605,373.656,-24.295,21.447,-41.968
C01475=1015.813,79.260,373.689,-24.295,21.446,-41.971
C01476=1015.815,78.921,373.721,-24.295,21.448,-41.973
C01477=1015.815,78.588,373.753,-24.294,21.447,-41.977
C01478=1015.816,78.260,373.784,-24.293,21.448,-41.980
C01479=1015.818,77.935,373.815,-24.293,21.448,-41.984
C01480=1015.819,77.612,373.847,-24.292,21.448,-41.987
C01481=1015.820,77.289,373.878,-24.292,21.449,-41.990
C01482=1015.821,76.962,373.908,-24.292,21.449,-41.994
C01483=1015.822,76.632,373.940,-24.291,21.449,-41.997
C01484=1015.822,76.296,373.973,-24.291,21.449,-42.001
C01485=1015.824,75.954,374.004,-24.290,21.449,-42.004
C01486=1015.825,75.605,374.038,-24.290,21.450,-42.006
C01487=1015.826,75.250,374.072,-24.289,21.450,-42.010
C01488=1015.828,74.893,374.106,-24.289,21.450,-42.013
C01489=1015.829,74.536,374.140,-24.288,21.451,-42.017
C01490=1015.830,74.179,374.174,-24.288,21.451,-42.019
C01491=1015.831,73.823,374.208,-24.288,21.451,-42.023
C01492=1015.832,73.470,374.242,-24.287,21.452,-42.027
C01493=1015.833,73.119,374.275,-24.286,21.451,-42.030
C01494=1015.834,72.769,374.308,-24.286,21.452,-42.034
C01495=1015.835,72.421,374.341,-24.285,21.452,-42.037
C01496=1015.837,72.074,374.374,-24.285,21.453,-42.041
C01497=1015.837,71.730,374.407,-24.285,21.453,-42.043
C01498=1015.839,71.384,374.439,-24.284,21.453,-42.047
C01499=1015.840,71.040,374.471,-24.284,21.454,-42.051
C01500=1015.841,70.695,374.504,-24.283,21.453,-42.054
C01501=1015.842,70.351,374.537,-24.283,21.454,-42.058
C01502=1015.843,70.007,374.570,-24.282,21.454,-42.061
C01503=1015.844,69.663,374.602,-24.282,21.455,-42.063
C01504=1015.845,69.318,374.635,-24.281,21.455,-42.067
C01505=1015.846,68.976,374.668,-24.281,21.456,-42.071
C01506=1015.847,68.633,374.701,-24.280,21.455,-42.074
C01507=1015.848,68.291,374.732,-24.280,21.456,-42.078
C01508=1015.850,67.952,374.765,-24.279,21.456,-42.082
C01509=1015.850,67.612,374.796,-24.279,21.456,-42.085
C01510=1015.851,67.274,374.829,-24.279,21.457,-42.087
C01511=1015.852,66.936,374.860,-24.278,21.457,-42.091
C01512=1015.853,66.599,374.892,-24.278,21.457,-42.094
C01513=1015.855,66.264,374.924,-24.277,21.457,-42.098
C01514=1015.856,65.931,374.955,-24.277,21.458,-42.102
C01515=1015.856,65.592,374.987,-24.276,21.457,-42.105
C01516=1015.858,65.238,375.020,-24.276,21.459,-42.108
C01517=1015.859,64.861,375.056,-24.275,21.458,-42.113
C01518=1015.860,64.466,375.093,-24.274,21.459,-42.116
C01519=1015.861,64.079,375.129,-24.274,21.459,-42.120
C01520=1015.862,63.723,375.163,-24.274,21.460,-42.124
C01521=1015.865,63.350,375.196,-24.273,21.460,-42.128
C01522=1015.869,63.131,375.215,-24.273,21.461,-42.130
C01523=1015.872,62.907,375.235,-24.272,21.460,-42.131
C01524=1015.878,62.512,375.268,-24.272,21.460,-42.135
C01525=1015.884,62.175,375.298,-24.271,21.461,-42.139
C01526=1015.888,61.841,375.326,-24.271,21.461,-42.142
C01527=1015.894,61.506,375.355,-24.270,21.462,-42.146
C01528=1015.899,61.171,375.384,-24.270,21.461,-42.149
C01529=1015.904,60.836,375.413,-24.269,21.462,-42.153
C01530=1015.909,60.501,375.442,-24.269,21.462,-42.157
C01531=1015.914,60.166,375.470,-24.268,21.462,-42.160
C01532=1015.919,59.831,375.499,-24.268,21.463,-42.163
C01533=1015.923,59.496,375.528,-24.268,21.464,-42.166
C01534=1015.929,59.161,375.557,-24.267,21.464,-42.170
C01535=1015.934,58.826,375.586,-24.267,21.464,-42.173
C01536=1015.938,58.491,375.614,-24.266,21.464,-42.177
C01537=1015.944,58.156,375.644,-24.266,21.465,-42.181
C01538=1015.948,57.821,375.672,-24.265,21.464,-42.184
C01539=1015.953,57.486,375.701,-24.264,21.465,-42.188
C01540=1015.958,57.152,375.730,-24.264,21.465,-42.192
C01541=1015.962,56.816,375.759,-24.264,21.466,-42.194
C01542=1015.967,56.481,375.788,-24.263,21.466,-42.197
C01543=1015.972,56.146,375.816,-24.263,21.466,-42.201
C01544=1015.977,55.811,375.845,-24.262,21.467,-42.205
C01545=1015.982,55.476,375.873,-24.262,21.467,-42.209
C01546=1015.986,55.141,375.902,-24.261,21.467,-42.212
C01547=1015.991,54.806,375.931,-24.261,21.467,-42.216
C01548=1015.996,54.471,375.960,-24.260,21.468,-42.220
C01549=1016.000,54.136,375.989,-24.260,21.468,-42.223
C01550=1016.005,53.801,376.018,-24.259,21.468,-42.227
C01551=1016.010,53.466,376.046,-24.259,21.468,-42.230
C01552=1016.014,53.132,376.075,-24.258,21.469,-42.234
C01553=1016.019,52.797,376.103,-24.258,21.469,-42.238
C01554=1016.023,52.462,376.132,-24.257,21.470,-42.240
C01555=1016.028,52.126,376.161,-24.257,21.470,-42.244
C01556=1016.032,51.792,376.190,-24.256,21.470,-42.247
C01557=1016.037,51.457,376.218,-24.256,21.471,-42.251
C01558=1016.041,51.122,376.247,-24.255,21.471,-42.254
C01559=1016.045,50.787,376.276,-24.255,21.471,-42.258
C01560=1016.050,50.452,376.304,-24.254,21.471,-42.262
C01561=1016.054,50.117,376.333,-24.254,21.472,-42.266
C01562=1016.060,49.782,376.362,-24.253,21.472,-42.269
C01563=1016.063,49.447,376.391,-24.253,21.472,-42.273
C01564=1016.068,49.112,376.420,-24.252,21.473,-42.277
C01565=1016.072,48.777,376.448,-24.252,21.473,-42.280
C01566=1016.077,48.443,376.477,-24.251,21.473,-42.284
C01567=1016.081,48.107,376.505,-24.251,21.473,-42.287
C01568=1016.086,47.772,376.533,-24.250,21.474,-42.291
C01569=1016.090,47.437,376.562,-24.250,21.474,-42.295
C01570=1016.094,47.103,376.590,-24.249,21.475,-42.299
C01571=1016.098,46.767,376.619,-24.249,21.475,-42.302
C01572=1016.102,46.433,376.647,-24.248,21.475,-42.306
C01573=1016.107,46.098,376.676,-24.248,21.475,-42.309
C01574=1016.111,45.763,376.705,-24.247,21.476,-42.313
C01575=1016.115,45.428,376.733,-24.247,21.476,-42.317
C01576=1016.120,45.093,376.762,-24.246,21.477,-42.321
C01577=1016.123,44.759,376.791,-24.246,21.477,-42.325
C01578=1016.127,44.424,376.819,-24.245,21.477,-42.328
C01579=1016.132,44.089,376.848,-24.245,21.477,-42.332
C01580=1016.136,43.754,376.877,-24.244,21.478,-42.335
C01581=1016.139,43.419,376.905,-24.244,21.478,-42.339
C01582=1016.144,43.085,376.933,-24.243,21.479,-42.343
C01583=1016.148,42.749,376.962,-24.243,21.479,-42.347
C01584=1016.152,42.414,376.991,-24.242,21.479,-42.350
C01585=1016.156,42.080,377.019,-24.242,21.479,-42.354
C01586=1016.160,41.745,377.048,-24.241,21.480,-42.357
C01587=1016.164,41.410,377.076,-24.241,21.480,-42.361
C01588=1016.168,41.075,377.104,-24.240,21.481,-42.365
C01589=1016.172,40.740,377.133,-24.240,21.481,-42.369
C01590=1016.176,40.406,377.161,-24.239,21.481,-42.372
C01591=1016.181,40.071,377.190,-24.239,21.481,-42.376
C01592=1016.184,39.736,377.218,-24.238,21.482,-42.380
C01593=1016.188,39.401,377.246,-24.238,21.482,-42.383
C01594=1016.192,39.067,377.274,-24.237,21.483,-42.387
C01595=1016.196,38.732,377.304,-24.237,21.483,-42.391
C01596=1016.199,38.397,377.332,-24.236,21.483,-42.395
C01597=1016.203,38.063,377.360,-24.236,21.483,-42.398
C01598=1016.207,37.728,377.389,-24.235,21.484,-42.402
C01599=1016.211,37.393,377.417,-24.235,21.484,-42.405
C01600=1016.215,37.058,377.445,-24.234,21.485,-42.409
C01601=1016.219,36.723,377.474,-24.234,21.485,-42.413
C01602=1016.222,36.389,377.502,-24.233,21.485,-42.418
C01603=1016.226,36.054,377.530,-24.232,21.485,-42.422
C01604=1016.230,35.720,377.559,-24.232,21.486,-42.426
C01605=1016.234,35.385,377.587,-24.231,21.485,-42.429
C01606=1016.237,35.050,377.615,-24.231,21.486,-42.433
C01607=1016.240,34.716,377.643,-24.230,21.486,-42.437
C01608=1016.245,34.381,377.672,-24.230,21.487,-42.440
C01609=1016.248,34.046,377.700,-24.229,21.487,-42.444
C01610=1016.252,33.712,377.729,-24.229,21.488,-42.448
C01611=1016.255,33.378,377.757,-24.228,21.488,-42.452
C01612=1016.259,33.043,377.785,-24.228,21.489,-42.455
C01613=1016.262,32.708,377.813,-24.227,21.489,-42.459
C01614=1016.266,32.374,377.841,-24.226,21.489,-42.464
C01615=1016.269,32.039,377.870,-24.226,21.489,-42.468
C01616=1016.273,31.705,377.898,-24.225,21.489,-42.471
C01617=1016.276,31.370,377.926,-24.225,21.490,-42.475
C01618=1016.280,31.035,377.954,-24.224,21.490,-42.479
C01619=1016.284,30.701,377.982,-24.224,21.491,-42.483
C01620=1016.286,30.367,378.011,-24.223,21.491,-42.486
C01621=1016.290,30.032,378.039,-24.223,21.492,-42.490
C01622=1016.294,29.698,378.067,-24.222,21.492,-42.494
C01623=1016.297,29.363,378.095,-24.222,21.493,-42.498
C01624=1016.301,29.029,378.124,-24.221,21.492,-42.503
C01625=1016.304,28.694,378.152,-24.221,21.493,-42.507
C01626=1016.307,28.360,378.180,-24.220,21.493,-42.510
C01627=1016.311,28.025,378.208,-24.220,21.494,-42.514
C01628=1016.314,27.691,378.236,-24.219,21.494,-42.518
C01629=1016.318,27.357,378.264,-24.219,21.495,-42.522
C01630=1016.320,27.022,378.292,-24.218,21.494,-42.525
C01631=1016.324,26.688,378.321,-24.217,21.494,-42.530
C01632=1016.327,26.354,378.349,-24.217,21.495,-42.534
C01633=1016.330,26.019,378.376,-24.216,21.495,-42.538
C01634=1016.333,25.686,378.405,-24.216,21.496,-42.541
C01635=1016.337,25.351,378.433,-24.215,21.496,-42.545
C01636=1016.340,25.016,378.461,-24.215,21.497,-42.549
C01637=1016.343,24.683,378.489,-24.214,21.497,-42.553
C01638=1016.346,24.348,378.517,-24.213,21.497,-42.558
C01639=1016.349,24.022,378.545,-24.213,21.498,-42.560
C01640=1016.352,23.727,378.570,-24.213,21.498,-42.562
C01641=1016.354,23.476,378.590,-24.212,21.498,-42.565
C01642=1016.358,23.067,378.624,-24.211,21.499,-42.573
C01643=1016.362,22.658,378.659,-24.210,21.499,-42.580
C01644=1016.364,22.405,378.679,-24.210,21.500,-42.582
C01645=1016.367,22.110,378.704,-24.210,21.501,-42.584
C01646=1016.370,21.787,378.731,-24.209,21.500,-42.588
C01647=1016.373,21.430,378.761,-24.209,21.501,-42.593
C01648=1016.375,21.223,378.778,-24.208,21.501,-42.597
C01649=1016.377,20.995,378.797,-24.208,21.502,-42.599
C01650=1016.379,20.754,378.818,-24.208,21.502,-42.601
C01651=1016.381,20.506,378.839,-24.207,21.502,-42.603
C01652=1016.383,20.259,378.859,-24.207,21.502,-42.604
C01653=1016.385,20.023,378.879,-24.207,21.502,-42.608
C01654=1016.389,19.606,378.913,-24.206,21.503,-42.613
C01655=1016.392,19.257,378.943,-24.205,21.502,-42.619
C01656=1016.395,18.926,378.971,-24.205,21.503,-42.622
C01657=1016.399,18.594,378.998,-24.204,21.503,-42.626
C01658=1016.401,18.263,379.025,-24.204,21.504,-42.630
C01659=1016.404,17.932,379.054,-24.203,21.504,-42.634
C01660=1016.406,17.601,379.080,-24.202,21.504,-42.639
C01661=1016.409,17.272,379.108,-24.202,21.505,-42.643
C01662=1016.412,16.942,379.135,-24.201,21.505,-42.646
C01663=1016.414,16.614,379.163,-24.201,21.506,-42.650
C01664=1016.417,16.285,379.190,-24.200,21.506,-42.654
C01665=1016.420,15.958,379.218,-24.200,21.507,-42.658
C01666=1016.423,15.631,379.244,-24.199,21.507,-42.663
C01667=1016.425,15.305,379.272,-24.199,21.507,-42.667
C01668=1016.428,14.979,379.299,-24.198,21.508,-42.670
C01669=1016.431,14.653,379.325,-24.198,21.508,-42.674
C01670=1016.434,14.328,379.353,-24.197,21.509,-42.678
C01671=1016.436,14.004,379.379,-24.197,21.509,-42.682
C01672=1016.438,13.679,379.406,-24.196,21.509,-42.687
C01673=1016.441,13.355,379.434,-24.195,21.509,-42.691
C01674=1016.444,13.032,379.461,-24.195,21.510,-42.694
C01675=1016.447,12.708,379.487,-24.194,21.510,-42.698
C01676=1016.449,12.384,379.514,-24.194,21.511,-42.702
C01677=1016.451,12.061,379.540,-24.193,21.511,-42.707
C01678=1016.453,11.737,379.567,-24.193,21.511,-42.711
C01679=1016.456,11.414,379.594,-24.192,21.512,-42.715
C01680=1016.459,11.092,379.621,-24.192,21.512,-42.718
C01681=1016.461,10.772,379.647,-24.191,21.513,-42.722
C01682=1016.463,10.453,379.673,-24.191,21.513,-42.726
C01683=1016.466,10.135,379.700,-24.190,21.514,-42.730
C01684=1016.468,9.820,379.726,-24.190,21.514,-42.733
C01685=1016.470,9.506,379.752,-24.189,21.514,-42.738
C01686=1016.473,9.191,379.778,-24.188,21.515,-42.742
C01687=1016.475,8.875,379.804,-24.188,21.515,-42.746
C01688=1016.478,8.559,379.831,-24.187,21.516,-42.750
C01689=1016.479,8.241,379.856,-24.186,21.515,-42.755
C01690=1016.482,7.920,379.883,-24.186,21.516,-42.759
C01691=1016.484,7.597,379.910,-24.186,21.516,-42.762
C01692=1016.486,7.272,379.936,-24.185,21.517,-42.766
C01693=1016.488,6.944,379.963,-24.185,21.517,-42.770
C01694=1016.491,6.615,379.990,-24.184,21.518,-42.774
C01695=1016.493,6.287,380.017,-24.183,21.518,-42.779
C01696=1016.495,5.957,380.045,-24.183,21.518,-42.783
C01697=1016.498,5.627,380.071,-24.182,21.519,-42.786
C01698=1016.500,5.297,380.099,-24.181,21.518,-42.792
C01699=1016.502,4.966,380.126,-24.181,21.519,-42.795
C01700=1016.505,4.635,380.153,-24.180,21.519,-42.799
C01701=1016.506,4.304,380.180,-24.180,21.521,-42.803
C01702=1016.509,3.974,380.208,-24.179,21.520,-42.807
C01703=1016.511,3.661,380.233,-24.179,21.521,-42.810
C01704=1016.513,3.371,380.257,-24.179,21.521,-42.814
C01705=1016.514,3.102,380.279,-24.178,21.522,-42.818
C01706=1016.516,2.839,380.300,-24.177,21.522,-42.823
C01707=1016.518,2.571,380.322,-24.177,21.522,-42.827
C01708=1016.519,2.283,380.346,-24.176,21.523,-42.831
C01709=1016.522,1.971,380.371,-24.176,21.523,-42.834
C01710=1016.524,1.640,380.399,-24.175,21.523,-42.838
C01711=1016.526,1.307,380.426,-24.175,21.524,-42.842
C01712=1016.528,0.973,380.454,-24.174,21.525,-42.846
C01713=1016.530,0.638,380.480,-24.173,21.525,-42.851
C01714=1016.532,0.302,380.508,-24.173,21.525,-42.855
C01715=1016.534,-0.036,380.536,-24.172,21.526,-42.858
C01716=1016.535,-0.374,380.563,-24.172,21.526,-42.864
C01717=1016.538,-0.714,380.591,-24.171,21.526,-42.867
C01718=1016.540,-1.055,380.619,-24.170,21.527,-42.873
C01719=1016.542,-1.398,380.647,-24.170,21.527,-42.877
C01720=1016.544,-1.744,380.675,-24.169,21.528,-42.880
C01721=1016.546,-2.090,380.703,-24.169,21.528,-42.886
C01722=1016.548,-2.439,380.732,-24.168,21.529,-42.890
C01723=1016.550,-2.788,380.760,-24.167,21.529,-42.895
C01724=1016.552,-3.139,380.789,-24.167,21.529,-42.899
C01725=1016.554,-3.493,380.817,-24.166,21.529,-42.904
C01726=1016.556,-3.846,380.846,-24.166,21.531,-42.908
C01727=1016.558,-4.204,380.875,-24.165,21.530,-42.913
C01728=1016.560,-4.566,380.904,-24.164,21.531,-42.919
C01729=1016.562,-4.933,380.935,-24.164,21.532,-42.923
C01730=1016.564,-5.302,380.965,-24.163,21.532,-42.928
C01731=1016.565,-5.676,380.995,-24.163,21.533,-42.932
C01732=1016.567,-6.051,381.025,-24.162,21.533,-42.937
C01733=1016.569,-6.426,381.055,-24.161,21.533,-42.941
C01734=1016.571,-6.801,381.086,-24.160,21.534,-42.947
C01735=1016.574,-7.172,381.116,-24.160,21.534,-42.952
C01736=1016.575,-7.542,381.146,-24.159,21.535,-42.956
C01737=1016.577,-7.908,381.176,-24.158,21.535,-42.961
C01738=1016.579,-8.272,381.205,-24.158,21.536,-42.967
C01739=1016.581,-8.634,381.234,-24.157,21.536,-42.971
C01740=1016.582,-8.997,381.264,-24.156,21.536,-42.976
C01741=1016.584,-9.359,381.293,-24.156,21.537,-42.982
C01742=1016.586,-9.721,381.322,-24.155,21.538,-42.985
C01743=1016.588,-10.083,381.351,-24.154,21.538,-42.991
C01744=1016.589,-10.444,381.380,-24.154,21.539,-42.995
C01745=1016.591,-10.804,381.410,-24.153,21.539,-43.000
C01746=1016.592,-11.163,381.438,-24.152,21.539,-43.006
C01747=1016.594,-11.521,381.467,-24.152,21.540,-43.009
C01748=1016.595,-11.876,381.496,-24.151,21.540,-43.014
C01749=1016.597,-12.232,381.525,-24.151,21.541,-43.019
C01750=1016.598,-12.586,381.553,-24.150,21.541,-43.024
C01751=1016.600,-12.937,381.581,-24.149,21.542,-43.028
C01752=1016.602,-13.287,381.609,-24.149,21.542,-43.033
C01753=1016.603,-13.636,381.637,-24.148,21.543,-43.037
C01754=1016.604,-13.982,381.665,-24.147,21.543,-43.042
C01755=1016.606,-14.327,381.693,-24.147,21.544,-43.046
C01756=1016.607,-14.669,381.720,-24.146,21.544,-43.052
C01757=1016.608,-15.008,381.748,-24.146,21.544,-43.055
C01758=1016.609,-15.347,381.775,-24.145,21.545,-43.061
C01759=1016.612,-15.683,381.802,-24.145,21.546,-43.065
C01760=1016.612,-16.018,381.828,-24.144,21.546,-43.070
C01761=1016.614,-16.353,381.856,-24.143,21.546,-43.074
C01762=1016.615,-16.686,381.882,-24.142,21.547,-43.079
C01763=1016.616,-17.020,381.909,-24.142,21.547,-43.083
C01764=1016.618,-17.353,381.935,-24.141,21.547,-43.088
C01765=1016.619,-17.686,381.962,-24.141,21.548,-43.092
C01766=1016.620,-18.050,381.991,-24.140,21.549,-43.100
C01767=1016.621,-18.272,382.008,-24.139,21.548,-43.103
C01768=1016.622,-18.519,382.029,-24.139,21.549,-43.105
C01769=1016.622,-18.781,382.049,-24.139,21.550,-43.107
C01770=1016.623,-19.043,382.070,-24.139,21.550,-43.109
C01771=1016.624,-19.291,382.090,-24.138,21.550,-43.112
C01772=1016.625,-19.707,382.123,-24.137,21.550,-43.118
C01773=1016.626,-19.880,382.137,-24.137,21.551,-43.122
C01774=1016.628,-20.213,382.163,-24.136,21.551,-43.127
C01775=1016.628,-20.545,382.190,-24.136,21.552,-43.131
C01776=1016.629,-20.878,382.217,-24.135,21.553,-43.135
C01777=1016.631,-21.211,382.243,-24.134,21.552,-43.140
C01778=1016.631,-21.544,382.269,-24.134,21.553,-43.144
C01779=1016.633,-21.877,382.296,-24.133,21.554,-43.149
C01780=1016.633,-22.209,382.322,-24.133,21.554,-43.153
C01781=1016.634,-22.542,382.349,-24.132,21.554,-43.158
C01782=1016.635,-22.875,382.375,-24.131,21.556,-43.162
C01783=1016.637,-23.207,382.401,-24.131,21.555,-43.168
C01784=1016.638,-23.540,382.427,-24.130,21.556,-43.171
C01785=1016.639,-23.873,382.454,-24.129,21.556,-43.177
C01786=1016.640,-24.206,382.480,-24.129,21.557,-43.181
C01787=1016.640,-24.538,382.506,-24.128,21.557,-43.186
C01788=1016.641,-24.871,382.533,-24.128,21.558,-43.190
C01789=1016.642,-25.204,382.559,-24.127,21.558,-43.195
C01790=1016.643,-25.537,382.586,-24.126,21.559,-43.199
C01791=1016.644,-25.870,382.612,-24.126,21.559,-43.204
C01792=1016.644,-26.202,382.638,-24.125,21.559,-43.208
C01793=1016.645,-26.535,382.664,-24.124,21.560,-43.214
C01794=1016.646,-26.868,382.691,-24.124,21.560,-43.217
C01795=1016.647,-27.201,382.717,-24.123,21.560,-43.223
C01796=1016.648,-27.533,382.743,-24.123,21.562,-43.227
C01797=1016.648,-27.866,382.769,-24.122,21.562,-43.232
C01798=1016.650,-28.199,382.796,-24.121,21.562,-43.236
C01799=1016.650,-28.532,382.822,-24.120,21.562,-43.241
C01800=1016.651,-28.864,382.848,-24.120,21.563,-43.245
C01801=1016.651,-29.198,382.874,-24.119,21.563,-43.250
C01802=1016.651,-29.531,382.900,-24.119,21.564,-43.254
C01803=1016.652,-29.863,382.927,-24.118,21.565,-43.260
C01804=1016.652,-30.196,382.953,-24.118,21.565,-43.264
C01805=1016.653,-30.529,382.978,-24.117,21.565,-43.269
C01806=1016.654,-30.861,383.005,-24.116,21.566,-43.273
C01807=1016.654,-31.194,383.031,-24.116,21.566,-43.278
C01808=1016.655,-31.527,383.057,-24.115,21.567,-43.282
C01809=1016.656,-31.859,383.083,-24.114,21.567,-43.287
C01810=1016.656,-32.192,383.109,-24.114,21.568,-43.291
C01811=1016.657,-32.525,383.135,-24.113,21.568,-43.296
C01812=1016.657,-32.858,383.161,-24.113,21.569,-43.301
C01813=1016.658,-33.190,383.187,-24.112,21.569,-43.306
C01814=1016.658,-33.523,383.214,-24.111,21.570,-43.310
C01815=1016.659,-33.856,383.239,-24.111,21.570,-43.315
C01816=1016.660,-34.188,383.265,-24.110,21.571,-43.319
C01817=1016.659,-34.521,383.291,-24.109,21.571,-43.324
C01818=1016.660,-34.854,383.317,-24.109,21.572,-43.328
C01819=1016.661,-35.186,383.343,-24.108,21.572,-43.334
C01820=1016.661,-35.519,383.369,-24.108,21.573,-43.337
